   "ComSd".Data.PlcOutputNormal."Q0.0" := "O_14VK1+SGV";
   "ComSd".Data.PlcOutputNormal."Q0.1" := "O_14VK2+SGV";
   "ComSd".Data.PlcOutputNormal."Q0.2" := "O_0VK1+SGV";
   "ComSd".Data.PlcOutputNormal."Q0.3" := "O_0VK2+SGV";
   "ComSd".Data.PlcOutputNormal."Q0.4" := "O_0VK3+SGV";
   "ComSd".Data.PlcOutputNormal."Q0.5" := "O_0VK4+SGV";
   "ComSd".Data.PlcOutputNormal."Q0.6" := "O_0F1.1+SGV";
   "ComSd".Data.PlcOutputNormal."Q0.7" := "O_0KA0.1+SGV";
   "ComSd".Data.PlcOutputNormal."Q1.0" := "O_0KA0.2+SGV";
   "ComSd".Data.PlcOutputNormal."Q1.1" := "O_0KA1+SGV";
   "ComSd".Data.PlcOutputNormal."Q1.2" := "O_8M1.T_c";
   "ComSd".Data.PlcOutputNormal."Q1.3" := "O_8M1.T_o";
   "ComSd".Data.PlcOutputNormal."Q1.4" := "O_8M1.L_c";
   "ComSd".Data.PlcOutputNormal."Q1.5" := "O_8M1.L_o";
   "ComSd".Data.PlcOutputNormal."Q1.6" := "O_8M1.R_c";
   "ComSd".Data.PlcOutputNormal."Q1.7" := "O_8M1.R_o";
   "ComSd".Data.PlcOutputNormal."Q2.0" := "O_8KA1+SGV";
   "ComSd".Data.PlcOutputNormal."Q2.1" := "O_8M1.B_l";
   "ComSd".Data.PlcOutputNormal."Q2.2" := "O_8M1.B_r";
   "ComSd".Data.PlcOutputNormal."Q2.3" := "O_2YV1/2.B+SGV";
   "ComSd".Data.PlcOutputNormal."Q2.4" := "O_2YV1.L+SGV";
   "ComSd".Data.PlcOutputNormal."Q2.5" := "O_2YV1.R+SGV";
   "ComSd".Data.PlcOutputNormal."Q2.6" := "O_5YV1+SGX";
   "ComSd".Data.PlcOutputNormal."Q2.7" := "O_spare27";
END_REGION

REGION Network 4 (SCL): Data PLC Output Safety

   "ComSd".Data.PlcOutputSafety."Q900.0" := "SO_safetynew";
   "ComSd".Data.PlcOutputSafety."Q900.1" := "SO_14HV1+SSTL/R";
   "ComSd".Data.PlcOutputSafety."Q900.2" := "SO_14KA1+SGV";
   "ComSd".Data.PlcOutputSafety."Q900.3" := "SO_14KA2+SGV";
   "ComSd".Data.PlcOutputSafety."Q908.0" := "SO_ST.3HF+SGV";
   "ComSd".Data.PlcOutputSafety."Q908.1" := "SO_ST.5HF+SGV";
   "ComSd".Data.PlcOutputSafety."Q908.2" := "SO_5AX1+SGX";
   "ComSd".Data.PlcOutputSafety."Q908.3" := "SO_spare9083";
END_REGION
END_FUNCTION_BLOCK

FUNCTION_BLOCK "ErrCom"   // FB303, FBD
{ S7_Optimized_Access := 'FALSE' }
// stored: AutoNumber false, SetENOAutomatically false
   VAR
      Var { S7_SetPoint := 'True'} : "TypeVar";
      T : Array[1..1] of IEC_TIMER;
   END_VAR
   VAR_TEMP
      ComOk : Bool;
      PwrOk : Bool;
      SiOk : Bool;
      EsOk : Bool;
      DoorOk : Bool;
   END_VAR
BEGIN

NETWORK
TITLE = general ok
// communication ok
      AN    "G".errComPc;
      =     #ComOk;

// power supply ok
      AN    "G"."errPs-0F1.1+SGV";
      =     #PwrOk;

// safety ok
      AN    "G".errSafetyModules;
      AN    "Si".aLaserErrFdb;
      AN    "Si".aAdjustmentErrFdb1;
      AN    "Si".aAdjustmentErrFdb2;
      =     #SiOk;

// doors ok
      A     #PwrOk;
      A     #SiOk;
      A     "Si".esInternal;
      =     #DoorOk;

// emergency ok
      A     #PwrOk;
      A     #SiOk;
      =     #EsOk;

REGION Network 2 (SCL): emergency stop

   // emergency stop internal (HMI)
   "ComErr".Err[2000] := #EsOk AND NOT "SI_14SB0/1+HMI" AND NOT "I_14SB0+HMI";
   "ComErr".Err[2001] := #EsOk AND NOT "SI_14SB0/1+HMI" AND NOT "I_14SB1+HMI";
   "ComErr".Err[2002] := #EsOk AND "Si".esInternalAckReq;

   // emergency stop external
   "ComErr".Err[2004] := #EsOk AND NOT "SI_NA_EXT+SGV";
   "ComErr".Err[2005] := #EsOk AND "Si".esExternalAckReq;
END_REGION

REGION Network 3 (SCL): safety doors

   // visual measurement - SGV
   "ComErr".Err[2010] := #DoorOk AND NOT "Si"."SGV-14SS1.TL".sig;
   "ComErr".Err[2011] := #DoorOk AND "Si"."SGV-14SS1.TL".sig AND NOT "Si"."SGV-14SS1.TL".ok;

   "ComErr".Err[2013] := #DoorOk AND NOT "Si"."SGV-14SS1.BL".sig;
   "ComErr".Err[2014] := #DoorOk AND "Si"."SGV-14SS1.BL".sig AND NOT "Si"."SGV-14SS1.BL".ok;

   "ComErr".Err[2016] := #DoorOk AND NOT "Si"."SGV-14SS1.TR".sig;
   "ComErr".Err[2017] := #DoorOk AND "Si"."SGV-14SS1.TR".sig AND NOT "Si"."SGV-14SS1.TR".ok;

   "ComErr".Err[2019] := #DoorOk AND NOT "Si"."SGV-14SS1.BR".sig;
   "ComErr".Err[2020] := #DoorOk AND "Si"."SGV-14SS1.BR".sig AND NOT "Si"."SGV-14SS1.BR".ok;

   // visual measurement - SGX
   "ComErr".Err[2030] := #DoorOk AND NOT "Si"."SGX-14SS1.TL".sig;
   "ComErr".Err[2031] := #DoorOk AND "Si"."SGX-14SS1.TL".sig AND NOT "Si"."SGX-14SS1.TL".ok;

   "ComErr".Err[2033] := #DoorOk AND NOT "Si"."SGX-14SS1.BL".sig;
   "ComErr".Err[2034] := #DoorOk AND "Si"."SGX-14SS1.BL".sig AND NOT "Si"."SGX-14SS1.BL".ok;

   "ComErr".Err[2036] := #DoorOk AND NOT "Si"."SGX-14SS1.TR".sig;
   "ComErr".Err[2037] := #DoorOk AND "Si"."SGX-14SS1.TR".sig AND NOT "Si"."SGX-14SS1.TR".ok;

   "ComErr".Err[2039] := #DoorOk AND NOT "Si"."SGX-14SS1.BR".sig;
   "ComErr".Err[2040] := #DoorOk AND "Si"."SGX-14SS1.BR".sig AND NOT "Si"."SGX-14SS1.BR".ok;
END_REGION

REGION Network 4 (SCL): manual

   // setting mode - SSTL
   "ComErr".Err[2050] := #ComOk AND #PwrOk AND #SiOk AND "Si".esInternal AND "Si".settingModeActive;

   // jog mode - SSTL
   "ComErr".Err[2052] := #ComOk AND #PwrOk AND #SiOk AND "Si".esInternal AND "Si".jogModeActive;

   // air-conditioning off - SSTR
   "ComErr".Err[2054] := #ComOk AND #PwrOk AND "I_0SH1+SSTR";
END_REGION

REGION Network 5 (SCL): safety

   // fault safety modules plc
   "ComErr".Err[2060] := #ComOk AND #PwrOk AND "G".errSafetyModules;

   // areas
   "ComErr".Err[2075] := #ComOk AND #PwrOk AND "SI_NA_EXT+SGV" AND  "SI_14SB0/1+HMI" AND (NOT "Si".esInternal OR NOT "Si".esExternal);

   // monitoring feedback
   "ComErr".Err[2080] := #ComOk AND #PwrOk AND "Si".aLaserErrFdb;
   "ComErr".Err[2081] := #ComOk AND #PwrOk AND "Si".aAdjustmentErrFdb1;
   "ComErr".Err[2082] := #ComOk AND #PwrOk AND "Si".aAdjustmentErrFdb2;
   "ComErr".Err[2083] := #ComOk AND #PwrOk AND  "G".Cfg.xrayActive AND "Si".aXrayErrFdb;
END_REGION

REGION Network 6 (SCL): fault sensor
   "ComErr".Err[2090] := "Sen"."1BTR2+SGV".err;
   "ComErr".Err[2091] := "Sen"."1BTR2+SGX".err;
END_REGION

REGION Network 7 (SCL): fault encoder
   "ComErr".Err[2100] := "Enc"."1BCI1".err;
   "ComErr".Err[2101] := "Enc"."1BCM1".err;
   "ComErr".Err[2102] := "Enc"."1BCO1".err;
END_REGION

REGION Network 8 (SCL): communication
   // fault watchdog
   "ComErr".Err[2110] := "G".errComPc;

   // release infeed
   "ComErr".Err[2111] := "G".errNoReleaseInf;
END_REGION

REGION Network 9 (SCL): fault general

   // power supply
   "ComErr".Err[2120] := "G"."errPs-0F1.1+SGV";

   // air conditioner
   "ComErr".Err[2121] := "G"."errAc-0E1+SGV";
   "ComErr".Err[2122] := "G"."errAc-0E2+SGX";
   "ComErr".Err[2123] := "G"."errAc-0E1.1+SGV";

   // err version
   "ComErr".Err[2125] := "G".errVersion;
END_REGION

REGION Network 10 (SCL): off information
   "ComErr".Err[2140] := "G".adjScannerOff;
   "ComErr".Err[2141] := "G".adjTopOff;
   "ComErr".Err[2142] := "G".adjLeftOff;
   "ComErr".Err[2143] := "G".adjRightOff;
   "ComErr".Err[2144] := "G".air1Off;
   "ComErr".Err[2145] := "G".air2Off;
   "ComErr".Err[2146] := "G".airXrayOff;
   "ComErr".Err[2147] := "G".airDehOff;
END_REGION

REGION Network 11 (SCL): fault adjustment

   // adjustment scannerhousing (-8M1.B+SGV)
   "ComErr".Err[2150] := "ComSd".Data.Scanner.Err;
   "ComErr".Err[2151] := "Enc"."8B1.B".err;
   "ComErr".Err[2152] := "Sen"."8S1.B".err;
   "ComErr".Err[2153] := "Sen"."8S2.B".err;
   "ComErr".Err[2154] := "Si".aAdjustment AND NOT "ComSd".Data.Scanner.refRun AND NOT "ComSd".Data.Scanner.refOk;
   "ComErr".Err[2155] := "Si".aAdjustment AND "ComSd".Data.Scanner.refRun;
   "ComErr".Err[2156] := "Si".aAdjustment AND "AdjScanner_DB".Cmd.auto AND NOT"ComSd".Data.Scanner.PosOk;
   "ComErr".Err[2157] := "Si".aAdjustment AND "ComRd".Data.Scanner.ManModeActive;

   // adjustment metering bar top (-8M1.T+SGV)
   "ComErr".Err[2160] := "ComSd".Data.Top.Err;
   "ComErr".Err[2161] := "ComSd".Data.Top.ErrEnc;
   "ComErr".Err[2162] := "Sen"."8S1.T".err;
   "ComErr".Err[2163] := "Sen"."8S2.T".err;
   "ComErr".Err[2164] := "Si".aAdjustment AND NOT "ComSd".Data.Top.refRun AND NOT "ComSd".Data.Top.refOk;
   "ComErr".Err[2165] := "Si".aAdjustment AND "ComSd".Data.Top.refRun;
   "ComErr".Err[2166] := "Si".aAdjustment AND "AdjTop_DB".Cmd.auto AND ((NOT "G".Cfg.adjTopActiveLinMot AND "Enc"."8BC1.T".notInPos) OR ("G".Cfg.adjTopActiveLinMot AND "Enc"."8U1.T".notInPos));
   "ComErr".Err[2167] := "Si".aAdjustment AND "ComRd".Data.Top.ManModeActive;

   // adjustment metering bar left (-8M1.L+SGV)
   "ComErr".Err[2170] := "ComSd".Data.Left.Err;
   "ComErr".Err[2171] := "ComSd".Data.Left.ErrEnc;
   "ComErr".Err[2172] := "Sen"."8S1.L".err;
   "ComErr".Err[2173] := "Sen"."8S2.L".err;
   "ComErr".Err[2174] := "Si".aAdjustment AND NOT "ComSd".Data.Left.refRun AND NOT "ComSd".Data.Left.refOk;
   "ComErr".Err[2175] := "Si".aAdjustment AND "ComSd".Data.Left.refRun;
   "ComErr".Err[2176] := "Si".aAdjustment AND "AdjLeft_DB".Cmd.auto AND ((NOT "G".Cfg.adjLeftActiveLinMot AND "Enc"."8BC1.L".notInPos) OR ("G".Cfg.adjLeftActiveLinMot AND "Enc"."8U1.L".notInPos));
   "ComErr".Err[2177] := "Si".aAdjustment AND "ComRd".Data.Left.ManModeActive;

   // adjustment metering bar right (-8M1.R+SGV)
   "ComErr".Err[2180] := "ComSd".Data.Right.Err;
   "ComErr".Err[2181] := "ComSd".Data.Right.ErrEnc;
   "ComErr".Err[2182] := "Sen"."8S1.R".err;
   "ComErr".Err[2183] := "Sen"."8S2.R".err;
   "ComErr".Err[2184] := "Si".aAdjustment AND NOT "ComSd".Data.Right.refRun AND NOT "ComSd".Data.Right.refOk;
   "ComErr".Err[2185] := "Si".aAdjustment AND "ComSd".Data.Right.refRun;
   "ComErr".Err[2186] := "Si".aAdjustment AND "AdjRight_DB".Cmd.auto AND ((NOT "G".Cfg.adjRightActiveLinMot AND "Enc"."8BC1.R".notInPos) OR ("G".Cfg.adjRightActiveLinMot AND "Enc"."8U1.R".notInPos));
   "ComErr".Err[2187] := "Si".aAdjustment AND "ComRd".Data.Right.ManModeActive;

   // sensor for random adjustment
   "ComErr".Err[2190] := "Sen"."8B1".err AND "G".Cfg.adjTopActiveLinMot;
   "ComErr".Err[2191] := "Sen"."8B2".err AND "G".Cfg.adjLeftActiveLinMot;
   "ComErr".Err[2192] := "Sen"."8B3".err AND "G".Cfg.adjRightActiveLinMot;
END_REGION

REGION Network 12 (SCL): fault profinet

   // fault profinet
   "ComErr".Err[2200] := "Diag_DB".IoDataSys1.devices[1].error AND "G".Cfg.adjTopActiveLinMot;
   "ComErr".Err[2201] := "Diag_DB".IoDataSys1.devices[2].error AND "G".Cfg.adjLeftActiveLinMot;
   "ComErr".Err[2202] := "Diag_DB".IoDataSys1.devices[3].error AND "G".Cfg.adjRightActiveLinMot;
END_REGION
END_FUNCTION_BLOCK

FUNCTION_BLOCK "DataTakeOver"   // FB302, FBD
{ S7_Optimized_Access := 'TRUE' }
// stored: AutoNumber false, MemoryReserve 100, SetENOAutomatically false
   VAR
      Var { ExternalAccessible := 'False'; ExternalVisible := 'False'; ExternalWritable := 'False'} : "TypeVar";
   END_VAR
BEGIN

REGION Network 1 (SCL): config data from pc
   IF "ComRd".Data.Config.active AND "G".comOk THEN

       // config for mode
       "G".Cfg.adjScannerActive := "ComRd".Data.Config.adjScannerActive;
       "G".Cfg.adjTopActive := "ComRd".Data.Config.adjTopActive;
       "G".Cfg.adjLeftActive := "ComRd".Data.Config.adjLeftActive;
       "G".Cfg.adjRightActive := "ComRd".Data.Config.adjRightActive;

       "G".Cfg.adjTopActiveLinMot := "ComRd".Data.Config.adjTopLinMotActive;
       "G".Cfg.adjLeftActiveLinMot := "ComRd".Data.Config.adjLeftLinMotActive;
       "G".Cfg.adjRightActiveLinMot := "ComRd".Data.Config.adjRightLinMotActive;

       "G".Cfg.xrayActive := "ComRd".Data.Config.xrayActive ;

       // config for mode
       "G".Cfg.modeBoardPassing:= "ComRd".Data.Config.modeBoardPassing;
       "G".Cfg.modeDimension := "ComRd".Data.Config.modeDimension;
       "G".Cfg.modeRandomAdj := "ComRd".Data.Config.modeRandomAdj;

       // config for sensor for random adjustment
       IF "ComRd".Data.Config.modeDimension = 3 OR "ComRd".Data.Config.modeDimension = 4 THEN
           "G".Cfg.senTopActive := TRUE;
       ELSE
           "G".Cfg.senTopActive := FALSE;
       END_IF;
       IF "ComRd".Data.Config.modeDimension = 2 OR "ComRd".Data.Config.modeDimension = 4 THEN
           IF "ComRd".Data.Config.modeBoardPassing = 3 THEN
               "G".Cfg.senLeftActive := TRUE;
               "G".Cfg.senRightActive := TRUE;
           ELSIF "ComRd".Data.Config.modeBoardPassing = 2 THEN
               "G".Cfg.senLeftActive := TRUE;
               "G".Cfg.senRightActive := FALSE;
           ELSIF "ComRd".Data.Config.modeBoardPassing = 1 THEN
               "G".Cfg.senLeftActive := FALSE;
               "G".Cfg.senRightActive := TRUE;
           END_IF;
       ELSE
           "G".Cfg.senLeftActive := FALSE;
           "G".Cfg.senRightActive := FALSE;
       END_IF;

       // config for encoder 1
       IF "ComRd".Data.Config.enc1QuadEvalActive THEN
           "G".Cfg.enc1Gain := (1.0 / INT_TO_REAL("ComRd".Data.Config.enc1Factor)) * 1.0;
       ELSE
           "G".Cfg.enc1Gain := (1.0 / INT_TO_REAL("ComRd".Data.Config.enc1Factor)) * 1.0;
       END_IF;
       IF "ComRd".Data.Config.enc1Factor = -1 THEN
           "G".Cfg.enc1Active := FALSE;
       ELSE
           "G".Cfg.enc1Active := TRUE;
       END_IF;

   END_IF;
END_REGION

REGION Network 2 (SCL): batch from pc
   IF "G".comOk THEN
       // Width
       IF "ComRd".Data.batch.MinWidth = "ComRd".Data.batch.MaxWidth THEN
           "G".Batch.widthMin := DINT_TO_REAL("ComRd".Data.batch.MinWidth) / 10.0;
           "G".Batch.widthMax := DINT_TO_REAL("ComRd".Data.batch.MaxWidth) / 10.0;
           "G".Batch.width := DINT_TO_REAL("ComRd".Data.batch.MinWidth) / 10.0;
       ELSIF "ComRd".Data.batch.MinWidth <> "ComRd".Data.batch.MaxWidth THEN
           "G".Batch.widthMin := DINT_TO_REAL("ComRd".Data.batch.MinWidth) / 10.0;
           "G".Batch.widthMax := DINT_TO_REAL("ComRd".Data.batch.MaxWidth) / 10.0;
           "G".Batch.width := DINT_TO_REAL(("ComRd".Data.batch.MinWidth + "ComRd".Data.batch.MaxWidth) / 2) / 10.0;
       END_IF;

       // Thickness
       IF "ComRd".Data.batch.MinThickness = "ComRd".Data.batch.MaxThickness THEN
           "G".Batch.thicknessMin := DINT_TO_REAL("ComRd".Data.batch.MinThickness) / 10.0;
           "G".Batch.thicknessMax := DINT_TO_REAL("ComRd".Data.batch.MaxThickness) / 10.0;
           "G".Batch.thickness := DINT_TO_REAL("ComRd".Data.batch.MinThickness) / 10.0;
       ELSIF "ComRd".Data.batch.MinThickness <> "ComRd".Data.batch.MaxThickness THEN
           "G".Batch.thicknessMin := DINT_TO_REAL("ComRd".Data.batch.MinThickness) / 10.0;
           "G".Batch.thicknessMax := DINT_TO_REAL("ComRd".Data.batch.MaxThickness) / 10.0;
           "G".Batch.thickness := DINT_TO_REAL(("ComRd".Data.batch.MinThickness + "ComRd".Data.batch.MaxThickness) / 2) / 10.0;
       END_IF;
   END_IF;
END_REGION
END_FUNCTION_BLOCK

FUNCTION_BLOCK "Sensors"   // FB505, FBD
{ S7_Optimized_Access := 'TRUE' }
// stored: AutoNumber false, MemoryReserve 100, SetENOAutomatically false
   VAR
      Var { ExternalAccessible := 'False'; ExternalVisible := 'False'; ExternalWritable := 'False'} : "TypeVar";
      Enc { ExternalAccessible := 'False'; ExternalVisible := 'False'; ExternalWritable := 'False'} : Array[1..3] of "SysCounterFast";
      S { ExternalAccessible := 'False'; ExternalVisible := 'False'; ExternalWritable := 'False'} : Array[1..5] of "SysSensor";
      SIO { ExternalAccessible := 'False'; ExternalVisible := 'False'; ExternalWritable := 'False'} : Array[1..3] of "SysWenglorP3PC301";
      senRightEncAct { ExternalAccessible := 'False'; ExternalVisible := 'False'; ExternalWritable := 'False'} : Real;
      senRightValSmoth { ExternalAccessible := 'False'; ExternalVisible := 'False'; ExternalWritable := 'False'} : Real;
      senRightCntr { ExternalAccessible := 'False'; ExternalVisible := 'False'; ExternalWritable := 'False'} : DInt;
      senRightSum { ExternalAccessible := 'False'; ExternalVisible := 'False'; ExternalWritable := 'False'} : Real;
      senLeftEncAct { ExternalAccessible := 'False'; ExternalVisible := 'False'; ExternalWritable := 'False'} : Real;
      senLeftValSmoth { ExternalAccessible := 'False'; ExternalVisible := 'False'; ExternalWritable := 'False'} : Real;
      senLeftCntr { ExternalAccessible := 'False'; ExternalVisible := 'False'; ExternalWritable := 'False'} : DInt;
      senLeftSum { ExternalAccessible := 'False'; ExternalVisible := 'False'; ExternalWritable := 'False'} : Real;
      senTopEncAct { ExternalAccessible := 'False'; ExternalVisible := 'False'; ExternalWritable := 'False'} : Real;
      senTopValSmoth { ExternalAccessible := 'False'; ExternalVisible := 'False'; ExternalWritable := 'False'} : Real;
      senTopCntr { ExternalAccessible := 'False'; ExternalVisible := 'False'; ExternalWritable := 'False'} : DInt;
      senTopSum { ExternalAccessible := 'False'; ExternalVisible := 'False'; ExternalWritable := 'False'} : Real;
      deltaSaved { ExternalAccessible := 'False'; ExternalVisible := 'False'; ExternalWritable := 'False'} : Real;
      senLeftValValid { ExternalAccessible := 'False'; ExternalVisible := 'False'; ExternalWritable := 'False'} : Bool;
      senRightValValid { ExternalAccessible := 'False'; ExternalVisible := 'False'; ExternalWritable := 'False'} : Bool;
      senTopValValid { ExternalAccessible := 'False'; ExternalVisible := 'False'; ExternalWritable := 'False'} : Bool;
      widthMeasureOk { ExternalAccessible := 'False'; ExternalVisible := 'False'; ExternalWritable := 'False'} : Bool;
   END_VAR
   VAR_TEMP
      tempMin : Real;
      tempMax : Real;
      tempWidth : Real;
   END_VAR
   VAR_TEMP   // added for the SCL form of the ladder/FBD networks
      _w1 : Bool;
   END_VAR
BEGIN

REGION Network 1: encoder infeed scanner
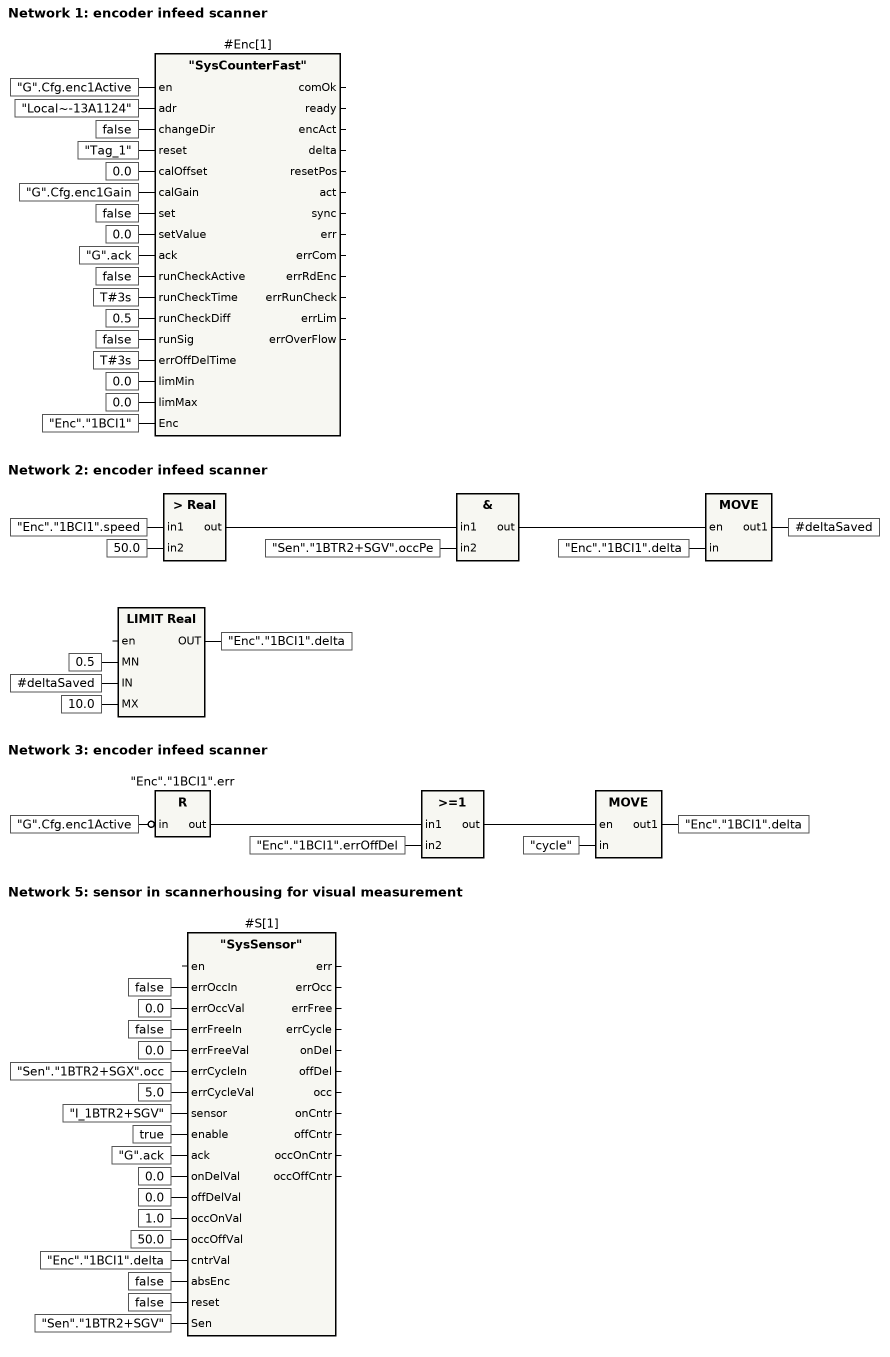
   IF "G".Cfg.enc1Active THEN
       #Enc[1](adr := "Local~-13A1124",   // "SysCounterFast"
               changeDir := false,
               reset := "Tag_1",
               calOffset := 0.0,
               calGain := "G".Cfg.enc1Gain,
               set := false,
               setValue := 0.0,
               ack := "G".ack,
               runCheckActive := false,
               runCheckTime := T#3s,
               runCheckDiff := 0.5,
               runSig := false,
               errOffDelTime := T#3s,
               limMin := 0.0,
               limMax := 0.0,
               Enc := "Enc"."1BCI1");
   END_IF;
END_REGION

REGION Network 2: encoder infeed scanner
   IF ("Enc"."1BCI1".speed > 50.0) AND "Sen"."1BTR2+SGV".occPe THEN
       #deltaSaved := "Enc"."1BCI1".delta;
   END_IF;
   "Enc"."1BCI1".delta := LIMIT(MN := 0.5, IN := #deltaSaved, MX := 10.0);
END_REGION

REGION Network 3: encoder infeed scanner
   IF NOT "G".Cfg.enc1Active THEN "Enc"."1BCI1".err := FALSE; END_IF;
   IF NOT "G".Cfg.enc1Active OR "Enc"."1BCI1".errOffDel THEN "Enc"."1BCI1".delta := "cycle"; END_IF;
END_REGION

REGION Network 4: - sensor monitoring -
END_REGION

REGION Network 5: sensor in scannerhousing for visual measurement
   #S[1](errOccIn := false,   // "SysSensor"
         errOccVal := 0.0,
         errFreeIn := false,
         errFreeVal := 0.0,
         errCycleIn := "Sen"."1BTR2+SGX".occ,
         errCycleVal := 5.0,
         sensor := "I_1BTR2+SGV",
         enable := true,
         ack := "G".ack,
         onDelVal := 0.0,
         offDelVal := 0.0,
         occOnVal := 1.0,
         occOffVal := 50.0,
         cntrVal := "Enc"."1BCI1".delta,
         absEnc := false,
         reset := false,
         Sen := "Sen"."1BTR2+SGV");
END_REGION

REGION Network 6: sensor in scannerhousing for xray measurement
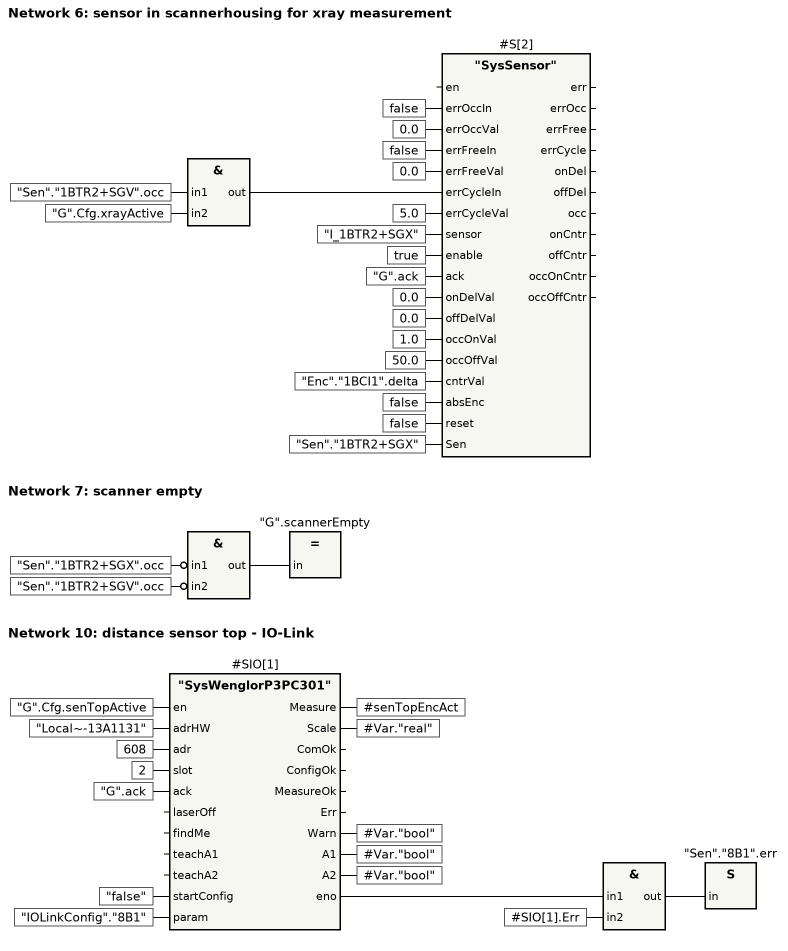
   #S[2](errOccIn := false,   // "SysSensor"
         errOccVal := 0.0,
         errFreeIn := false,
         errFreeVal := 0.0,
         errCycleIn := "Sen"."1BTR2+SGV".occ AND "G".Cfg.xrayActive,
         errCycleVal := 5.0,
         sensor := "I_1BTR2+SGX",
         enable := true,
         ack := "G".ack,
         onDelVal := 0.0,
         offDelVal := 0.0,
         occOnVal := 1.0,
         occOffVal := 50.0,
         cntrVal := "Enc"."1BCI1".delta,
         absEnc := false,
         reset := false,
         Sen := "Sen"."1BTR2+SGX");
END_REGION

REGION Network 7: scanner empty
   "G".scannerEmpty := NOT "Sen"."1BTR2+SGX".occ AND NOT "Sen"."1BTR2+SGV".occ;
END_REGION

REGION Network 8: distance sensor top
END_REGION

REGION Network 9 (SCL): distance sensor top - calibration value from pc
   "ComSd".Data.Measure.SetCalibratePosTopOk := FALSE;

   IF "ComRd".Data.Measure.SetCalibratePosTop THEN

       "Ref".senTopCalOffset := #senTopEncAct + "G".Batch.thickness;
       "ComSd".Data.Measure.SetCalibratePosTopOk := TRUE;
   END_IF;
END_REGION

REGION Network 10: distance sensor top - IO-Link
   #SIO[1](EN := "G".Cfg.senTopActive,   // "SysWenglorP3PC301"
           adrHW := "Local~-13A1131",
           adr := 608,
           slot := 2,
           ack := "G".ack,
           startConfig := "false",
           param := "IOLinkConfig"."8B1",
           Measure => #senTopEncAct,
           Scale => #Var."real",
           Warn => #Var."bool",
           A1 => #Var."bool",
           A2 => #Var."bool",
           ENO => #_w1);
   IF #_w1 AND #SIO[1].Err THEN "Sen"."8B1".err := TRUE; END_IF;
END_REGION

REGION Network 11 (SCL): distance sensor top - values
   IF "G".Cfg.senTopActive THEN
       IF #SIO[1].MeasureOk THEN
           "Sen"."8B1".val := "Ref".senTopCalOffset - #senTopEncAct;
       ELSE
           "Sen"."8B1".val := -50.0;
       END_IF;
       "ComSd".Data.Measure.ActValueTop := REAL_TO_DINT(#senTopEncAct * 10.0);

       IF "G".Cfg.modeBoardPassing = 3 THEN
           #tempMin := "G".Batch.widthMin / 4.0;
           #tempMax := "G".Batch.widthMax + 50.0;
       ELSE
           #tempMin := "G".Batch.widthMin / 2.0;
           #tempMax := "G".Batch.widthMax + 50.0;
       END_IF;
   ELSE
       #senTopEncAct :=  "Sen"."8B1".val := 0.0;
       "ComSd".Data.Measure.ActValueTop := 0;
   END_IF;
END_REGION

REGION Network 12: distance sensor top - occupied
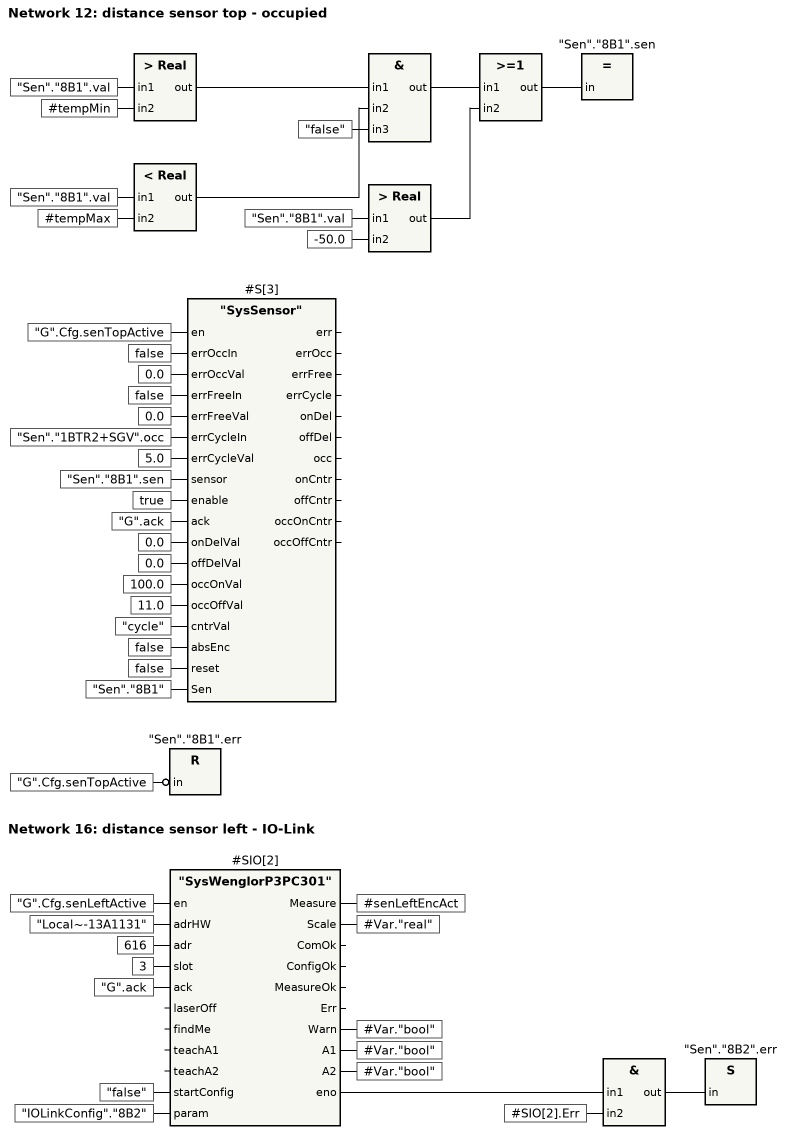
   "Sen"."8B1".sen := (("Sen"."8B1".val > #tempMin) AND ("Sen"."8B1".val < #tempMax) AND "false") OR ("Sen"."8B1".val > (-50.0));
   IF "G".Cfg.senTopActive THEN
       #S[3](errOccIn := false,   // "SysSensor"
             errOccVal := 0.0,
             errFreeIn := false,
             errFreeVal := 0.0,
             errCycleIn := "Sen"."1BTR2+SGV".occ,
             errCycleVal := 5.0,
             sensor := "Sen"."8B1".sen,
             enable := true,
             ack := "G".ack,
             onDelVal := 0.0,
             offDelVal := 0.0,
             occOnVal := 100.0,
             occOffVal := 11.0,
             cntrVal := "cycle",
             absEnc := false,
             reset := false,
             Sen := "Sen"."8B1");
   END_IF;
   IF NOT "G".Cfg.senTopActive THEN "Sen"."8B1".err := FALSE; END_IF;
END_REGION

REGION Network 13 (SCL): distance sensor top - smoothed value
   IF "Sen"."8B1".occPe THEN
       #senTopCntr := 10;
       #senTopSum := 0.0;
       #senTopValValid := false;
   ELSIF NOT "Sen"."8B1".occ OR #senTopCntr > 10 THEN
       #senTopCntr := 0;
   END_IF;

   IF "Sen"."8B1".occNe THEN
       #senTopValValid := false;
   END_IF;

   IF #senTopCntr > 0 AND "Sen"."8B1".sen THEN
       #senTopSum += "Sen"."8B1".val;
       #senTopCntr -= 1;
       IF #senTopCntr = 0 THEN
           #senTopValSmoth := #senTopSum / 10.0;
           #senTopValValid := true;
       END_IF;
   END_IF;

   IF "ComRd".Data.status.Auto AND  "G".Cfg.senTopActive THEN
       "Sen"."8B1".val := #senTopValSmoth;
   END_IF;
END_REGION

REGION Network 14: distance sensor left
END_REGION

REGION Network 15 (SCL): distance sensor left - calibration value from pc
   "ComSd".Data.Measure.SetCalibratePosLeftOk := FALSE;

   IF "ComRd".Data.Measure.SetCalibratePosLeft THEN

       #tempWidth := "G".Batch.width;
       IF "G".Cfg.modeBoardPassing = 3 THEN
           #tempWidth := "G".Batch.width / 2.0;
       END_IF;
       "Ref".senLeftCalOffset := #senLeftEncAct + #tempWidth;

       "ComSd".Data.Measure.SetCalibratePosLeftOk := TRUE;
   END_IF;
END_REGION

REGION Network 16: distance sensor left - IO-Link
   #SIO[2](EN := "G".Cfg.senLeftActive,   // "SysWenglorP3PC301"
           adrHW := "Local~-13A1131",
           adr := 616,
           slot := 3,
           ack := "G".ack,
           startConfig := "false",
           param := "IOLinkConfig"."8B2",
           Measure => #senLeftEncAct,
           Scale => #Var."real",
           Warn => #Var."bool",
           A1 => #Var."bool",
           A2 => #Var."bool",
           ENO => #_w1);
   IF #_w1 AND #SIO[2].Err THEN "Sen"."8B2".err := TRUE; END_IF;
END_REGION

REGION Network 17 (SCL): distance sensor left - values
   IF "G".Cfg.senLeftActive THEN

       IF #SIO[2].MeasureOk THEN
           "Sen"."8B2".val := "Ref".senLeftCalOffset - #senLeftEncAct;
       ELSE
           "Sen"."8B2".val := -50.0;
       END_IF;
       "ComSd".Data.Measure.ActValueLeft := REAL_TO_DINT("Sen"."8B2".val * 10.0);

       IF "G".Cfg.modeBoardPassing = 3 THEN
           #tempMin := "G".Batch.widthMin / 4.0;
           #tempMax := "G".Batch.widthMax + 50.0;
       ELSE
           #tempMin := "G".Batch.widthMin / 2.0;
           #tempMax := "G".Batch.widthMax + 50.0;
       END_IF;
   ELSE
       #senLeftEncAct :=  "Sen"."8B2".val := 0.0;
       "ComSd".Data.Measure.ActValueLeft := 0;
   END_IF;
END_REGION

REGION Network 18: distance sensor left - occupied
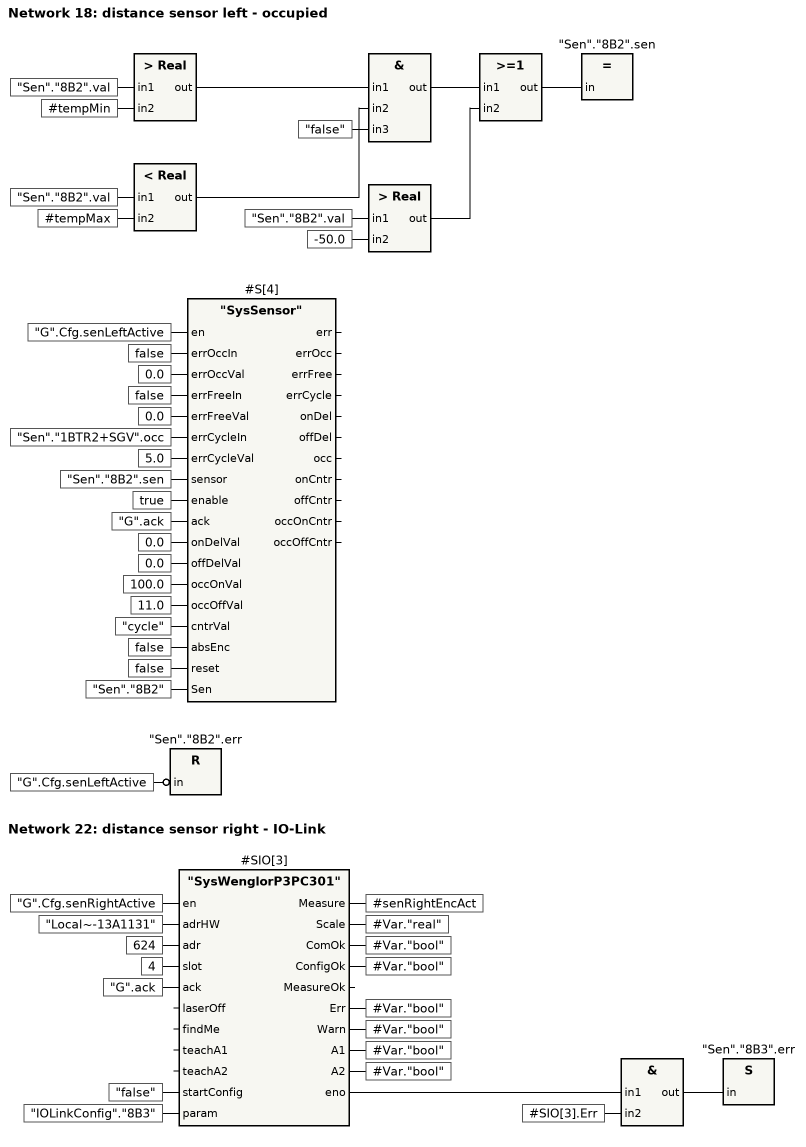
   "Sen"."8B2".sen := (("Sen"."8B2".val > #tempMin) AND ("Sen"."8B2".val < #tempMax) AND "false") OR ("Sen"."8B2".val > (-50.0));
   IF "G".Cfg.senLeftActive THEN
       #S[4](errOccIn := false,   // "SysSensor"
             errOccVal := 0.0,
             errFreeIn := false,
             errFreeVal := 0.0,
             errCycleIn := "Sen"."1BTR2+SGV".occ,
             errCycleVal := 5.0,
             sensor := "Sen"."8B2".sen,
             enable := true,
             ack := "G".ack,
             onDelVal := 0.0,
             offDelVal := 0.0,
             occOnVal := 100.0,
             occOffVal := 11.0,
             cntrVal := "cycle",
             absEnc := false,
             reset := false,
             Sen := "Sen"."8B2");
   END_IF;
   IF NOT "G".Cfg.senLeftActive THEN "Sen"."8B2".err := FALSE; END_IF;
END_REGION

REGION Network 19 (SCL): distance sensor left - smoothed value
   IF "Sen"."8B2".occPe THEN
       #senLeftCntr := 10;
       #senLeftSum := 0.0;
       #senLeftValValid := false;
   ELSIF NOT "Sen"."8B2".occ OR #senLeftCntr > 10 THEN
       #senLeftCntr := 0;
   END_IF;

   IF "Sen"."8B2".occNe THEN
       #senLeftValValid := false;
   END_IF;

   IF #senLeftCntr > 0 AND "Sen"."8B2".sen THEN
       #senLeftSum += "Sen"."8B2".val;
       #senLeftCntr -= 1;
       IF #senLeftCntr = 0 THEN
           #senLeftValSmoth := #senLeftSum / 10.0;
           #senLeftValValid := true;
       END_IF;
   END_IF;

   IF "ComRd".Data.status.Auto AND  "G".Cfg.senLeftActive THEN
       "Sen"."8B2".val := #senLeftValSmoth;
   END_IF;
END_REGION

REGION Network 20: distance sensor right
END_REGION

REGION Network 21 (SCL): distance sensor right - calibration value from pc
   "ComSd".Data.Measure.SetCalibratePosRightOk := FALSE;

   IF "ComRd".Data.Measure.SetCalibratePosRight THEN

       #tempWidth := "G".Batch.width;
       IF "G".Cfg.modeBoardPassing = 3 THEN
           #tempWidth := "G".Batch.width / 2.0;
       END_IF;
       "Ref".senRightCalOffset := #senRightEncAct + #tempWidth;

       "ComSd".Data.Measure.SetCalibratePosRightOk := TRUE;
   END_IF;
END_REGION

REGION Network 22: distance sensor right - IO-Link
   #SIO[3](EN := "G".Cfg.senRightActive,   // "SysWenglorP3PC301"
           adrHW := "Local~-13A1131",
           adr := 624,
           slot := 4,
           ack := "G".ack,
           startConfig := "false",
           param := "IOLinkConfig"."8B3",
           Measure => #senRightEncAct,
           Scale => #Var."real",
           ComOk => #Var."bool",
           ConfigOk => #Var."bool",
           Err => #Var."bool",
           Warn => #Var."bool",
           A1 => #Var."bool",
           A2 => #Var."bool",
           ENO => #_w1);
   IF #_w1 AND #SIO[3].Err THEN "Sen"."8B3".err := TRUE; END_IF;
END_REGION

REGION Network 23 (SCL): distance sensor right - values
   IF "G".Cfg.senRightActive THEN
       IF #SIO[3].MeasureOk THEN
           "Sen"."8B3".val := "Ref".senRightCalOffset - #senRightEncAct;
       ELSE
           "Sen"."8B3".val := -50.0;
       END_IF;
       "ComSd".Data.Measure.ActValueRight := REAL_TO_DINT("Sen"."8B3".val * 10.0);

       IF "G".Cfg.modeBoardPassing = 3 THEN
           #tempMin := "G".Batch.widthMin / 4.0;
           #tempMax := "G".Batch.widthMax + 50.0;
       ELSE
           #tempMin := "G".Batch.widthMin / 2.0;
           #tempMax := "G".Batch.widthMax + 50.0;
       END_IF;
   ELSE
       #senRightEncAct :=  "Sen"."8B3".val := 0.0;
       "ComSd".Data.Measure.ActValueRight := 0;
   END_IF;
END_REGION

REGION Network 24: distance sensor right - occupied
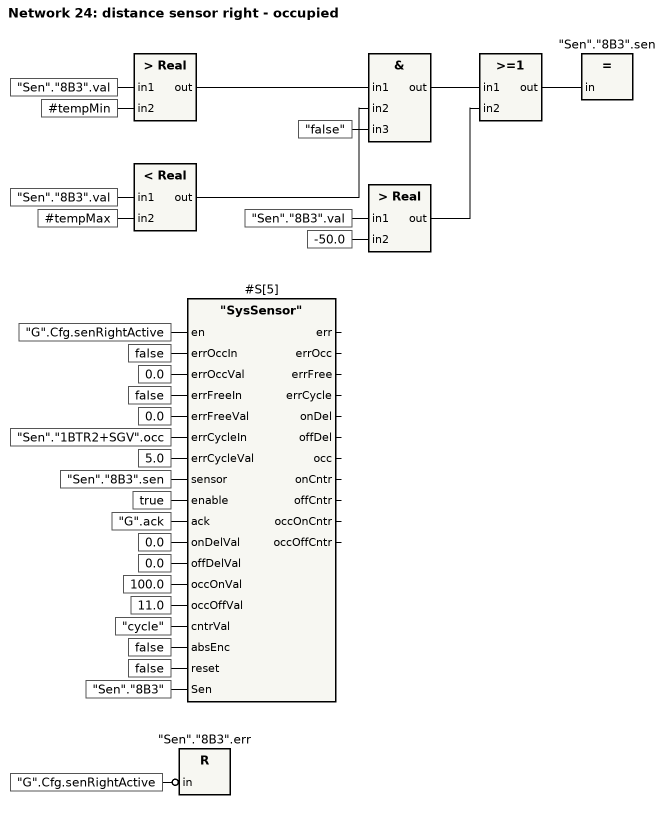
   "Sen"."8B3".sen := (("Sen"."8B3".val > #tempMin) AND ("Sen"."8B3".val < #tempMax) AND "false") OR ("Sen"."8B3".val > (-50.0));
   IF "G".Cfg.senRightActive THEN
       #S[5](errOccIn := false,   // "SysSensor"
             errOccVal := 0.0,
             errFreeIn := false,
             errFreeVal := 0.0,
             errCycleIn := "Sen"."1BTR2+SGV".occ,
             errCycleVal := 5.0,
             sensor := "Sen"."8B3".sen,
             enable := true,
             ack := "G".ack,
             onDelVal := 0.0,
             offDelVal := 0.0,
             occOnVal := 100.0,
             occOffVal := 11.0,
             cntrVal := "cycle",
             absEnc := false,
             reset := false,
             Sen := "Sen"."8B3");
   END_IF;
   IF NOT "G".Cfg.senRightActive THEN "Sen"."8B3".err := FALSE; END_IF;
END_REGION

REGION Network 25 (SCL): distance sensor right - smoothed value
   IF "Sen"."8B3".occPe THEN
       #senRightCntr := 10;
       #senRightSum := 0.0;
       #senRightValValid := false;
   ELSIF NOT "Sen"."8B3".occ OR #senRightCntr > 10 THEN
       #senRightCntr := 0;
   END_IF;

   IF "Sen"."8B3".occNe THEN
       #senRightValValid := false;
   END_IF;

   IF #senRightCntr > 0 AND "Sen"."8B3".sen THEN
       #senRightSum += "Sen"."8B3".val;
       #senRightCntr -= 1;
       IF #senRightCntr = 0 THEN
           #senRightValSmoth := #senRightSum / 10.0;
           #senRightValValid := true;
       END_IF;
   END_IF;

   IF "ComRd".Data.status.Auto AND  "G".Cfg.senRightActive THEN
       "Sen"."8B3".val := #senRightValSmoth;
   END_IF;
END_REGION

REGION Network 26 (SCL): distance sensor - data to pc
   // Thickness
   IF "G".Cfg.modeDimension = 3 OR "G".Cfg.modeDimension = 4 AND  NOT "Sen"."1BTR2+SGV".occ THEN
       "G".Batch.thicknessMeasure := "Sen"."8B1".val;
       // Version 5.13 - Dont look at min or max
       // IF "G".Batch.thicknessMeasure < "G".Batch.thicknessMin OR "G".Batch.thicknessMeasure > "G".Batch.thicknessMax  THEN
       //     "G".Batch.thicknessMeasure := "G".Batch.thickness;
       // END_IF;
       "ComSd".Data.Measure.Thickness := REAL_TO_DINT("G".Batch.thicknessMeasure * 10.0);
   ELSE
       "ComSd".Data.Measure.Thickness := 0;
   END_IF;

   // Width
   IF "G".Cfg.modeDimension = 2 OR "G".Cfg.modeDimension = 4 AND NOT "Sen"."1BTR2+SGV".occ  THEN
       #widthMeasureOk := false;
       IF "G".Cfg.modeBoardPassing = 1 AND  #senRightValValid  THEN
           "G".Batch.widthMeasure := "Sen"."8B3".val;
           #widthMeasureOk := true;
       ELSIF "G".Cfg.modeBoardPassing = 2 AND  #senLeftValValid THEN
           "G".Batch.widthMeasure := "Sen"."8B2".val;
           #widthMeasureOk := true;
       ELSIF "G".Cfg.modeBoardPassing = 3  AND #senLeftValValid  AND #senRightValValid  THEN
           "G".Batch.senLeftVal := "Sen"."8B2".val;
           "G".Batch.senRightVal := "Sen"."8B3".val;
           #widthMeasureOk := true;
           // Version 5.13 - Dont look at min or max
           // IF "G".Batch.senLeftVal < "G".Batch.widthMin / 2.0 - 50.0 OR "G".Batch.senLeftVal > "G".Batch.widthMax / 2.0 + 50.0 OR
           //     "G".Batch.senRightVal < "G".Batch.widthMin / 2.0 - 50.0 OR "G".Batch.senRightVal > "G".Batch.widthMax / 2.0 + 50.0 THEN
           //     "G".Batch.senLeftVal := "G".Batch.senRightVal := "G".Batch.width / 2.0;
           //     #widthMeasureOk := false;
           // END_IF;
           "G".Batch.widthMeasure := "G".Batch.senLeftVal + "G".Batch.senRightVal;
           "G".Batch.offsetBoard := ("G".Batch.senLeftVal - "G".Batch.senRightVal) / 2.0;
       END_IF;
       // Version 5.13 - Dont look at min or max
       // IF "G".Batch.widthMeasure < ("G".Batch.widthMin - 50.0)  OR "G".Batch.widthMeasure > ("G".Batch.widthMax + 50.0) THEN
       //     "G".Batch.widthMeasure := "G".Batch.width;
       //     #widthMeasureOk := false;
       // END_IF;
       "ComSd".Data.Measure.Width := REAL_TO_DINT(("G".Batch.widthMeasure) * 10.0);
   ELSE
       "ComSd".Data.Measure.Width := 0;
   END_IF;
END_REGION
END_FUNCTION_BLOCK

FUNCTION_BLOCK "SysCounterFast"   // FB2035, FBD
TITLE = manage a incremental encoder conected to a counter module
{ S7_Optimized_Access := 'TRUE' }
AUTHOR : MiCROTEC
VERSION : 1.6
// -2018.09 : Martin
// -2019.10 : Martin
// stored: AutoNumber false, MemoryReserve 100, SetENOAutomatically false
   VAR_INPUT
      adr { ExternalAccessible := 'False'; ExternalVisible := 'False'; ExternalWritable := 'False'} : HW_IO;   // I/O adresse
      changeDir { ExternalAccessible := 'False'; ExternalVisible := 'False'; ExternalWritable := 'False'} : Bool;   // change direction
      reset { ExternalAccessible := 'False'; ExternalVisible := 'False'; ExternalWritable := 'False'} : Bool;   // reset counter
      calOffset { ExternalAccessible := 'False'; ExternalVisible := 'False'; ExternalWritable := 'False'} : Real;   // offset [mm], the "Reset" will take effect after the offset value
      calGain { ExternalAccessible := 'False'; ExternalVisible := 'False'; ExternalWritable := 'False'} : Real;   // gain
      set { ExternalAccessible := 'False'; ExternalVisible := 'False'; ExternalWritable := 'False'} : Bool;   // set counter on "set value"
      setValue { ExternalAccessible := 'False'; ExternalVisible := 'False'; ExternalWritable := 'False'} : Real;   // set value [mm]
      ack { ExternalAccessible := 'False'; ExternalVisible := 'False'; ExternalWritable := 'False'} : Bool;   // fault acknowledge
      runCheckActive { ExternalAccessible := 'False'; ExternalVisible := 'False'; ExternalWritable := 'False'} : Bool;   // activate plausibility check of encoder value and run signal
      runCheckTime { ExternalAccessible := 'False'; ExternalVisible := 'False'; ExternalWritable := 'False'} : Time := T#3S;   // run signal check fault time
      runCheckDiff { ExternalAccessible := 'False'; ExternalVisible := 'False'; ExternalWritable := 'False'} : Real := 0.5;   // difference value for run check
      runSig { ExternalAccessible := 'False'; ExternalVisible := 'False'; ExternalWritable := 'False'} : Bool;   // run signal for drive
      errOffDelTime { ExternalAccessible := 'False'; ExternalVisible := 'False'; ExternalWritable := 'False'} : Time := T#1S;   // err off delayed time
      limMin { ExternalAccessible := 'False'; ExternalVisible := 'False'; ExternalWritable := 'False'} : Real;   // minimum limit position (0 = deactivated )
      limMax { ExternalAccessible := 'False'; ExternalVisible := 'False'; ExternalWritable := 'False'} : Real;   // maximum limit position (0 = deactivated )
   END_VAR
   VAR_OUTPUT
      comOk { ExternalAccessible := 'False'; ExternalVisible := 'False'; ExternalWritable := 'False'} : Bool;   // communication ok/active
      ready { ExternalAccessible := 'False'; ExternalVisible := 'False'; ExternalWritable := 'False'} : Bool;   // ready to work
      encAct { ExternalAccessible := 'False'; ExternalVisible := 'False'; ExternalWritable := 'False'} : DInt;   // actual position from counter
      delta { ExternalAccessible := 'False'; ExternalVisible := 'False'; ExternalWritable := 'False'} : Real;   // delta in millimeter
      resetPos { ExternalAccessible := 'False'; ExternalVisible := 'False'; ExternalWritable := 'False'} : Real;   // last reset position for the encoder value (ex. division sensor)
      act { ExternalAccessible := 'False'; ExternalVisible := 'False'; ExternalWritable := 'False'} : Real;   // actual position in millimeter
      sync { ExternalAccessible := 'False'; ExternalVisible := 'False'; ExternalWritable := 'False'} : Bool;   // reset puls (division sensor, or generate with offset)
      err { ExternalAccessible := 'False'; ExternalVisible := 'False'; ExternalWritable := 'False'} : Bool;   // fault
      errCom { ExternalAccessible := 'False'; ExternalVisible := 'False'; ExternalWritable := 'False'} : Bool;   // fault communication
      errRdEnc { ExternalAccessible := 'False'; ExternalVisible := 'False'; ExternalWritable := 'False'} : Bool;   // fault encoder from count module
      errRunCheck { ExternalAccessible := 'False'; ExternalVisible := 'False'; ExternalWritable := 'False'} : Bool;   // fault plausibility check run-signal/encoder-value
      errLim { ExternalAccessible := 'False'; ExternalVisible := 'False'; ExternalWritable := 'False'} : Bool;   // fault position is outside from limits
      errOverFlow { ExternalAccessible := 'False'; ExternalVisible := 'False'; ExternalWritable := 'False'} : Bool;   // fault implausible change in encoder value detected (maybe overflow or underflow)
   END_VAR
   VAR_IN_OUT
      Enc : "TypeEncoder";
   END_VAR
   VAR
      var { ExternalAccessible := 'False'; ExternalVisible := 'False'; ExternalWritable := 'False'; S7_SetPoint := 'True'} : "TypeVar";
      T { ExternalAccessible := 'False'; ExternalVisible := 'False'; ExternalWritable := 'False'; S7_SetPoint := 'True'} : Array[1..3] of IEC_TIMER;
      Rd { ExternalAccessible := 'False'; ExternalVisible := 'False'; ExternalWritable := 'False'} : Struct
         cntBit24 : Bool;   // count value
         stsDI1 : Bool;   // DI1 status
         stsDir : Bool;   // direction
         stsDI0 : Bool;   // DI0 status
         err : Bool;   // fault
         stsDI2 : Bool;   // Tm Count: status DI2
         stsReady : Bool;   // ready
         Wd : Bool;   // watchdog if used isochronous mode
         cntValue2 : Byte;   // count value
         cntValue : Word;   // count value
      END_STRUCT;
      encActOld { ExternalAccessible := 'False'; ExternalVisible := 'False'; ExternalWritable := 'False'} : DInt;
      deltaIncOld { ExternalAccessible := 'False'; ExternalVisible := 'False'; ExternalWritable := 'False'} : DInt;
      actualNoOffset { ExternalAccessible := 'False'; ExternalVisible := 'False'; ExternalWritable := 'False'} : Real;
      errLimMin { ExternalAccessible := 'False'; ExternalVisible := 'False'; ExternalWritable := 'False'} : Bool;
      errLimMax { ExternalAccessible := 'False'; ExternalVisible := 'False'; ExternalWritable := 'False'} : Bool;
   END_VAR
   VAR_TEMP
      tempDelta1 : DInt;
      tempRdRetVal : Int;
      tempErrOverFlow : Bool;
   END_VAR
   VAR_TEMP   // added for the SCL form of the ladder/FBD networks
      _w1 : Bool;
      _w2 : Bool;
   END_VAR
BEGIN

REGION Network 1: exit
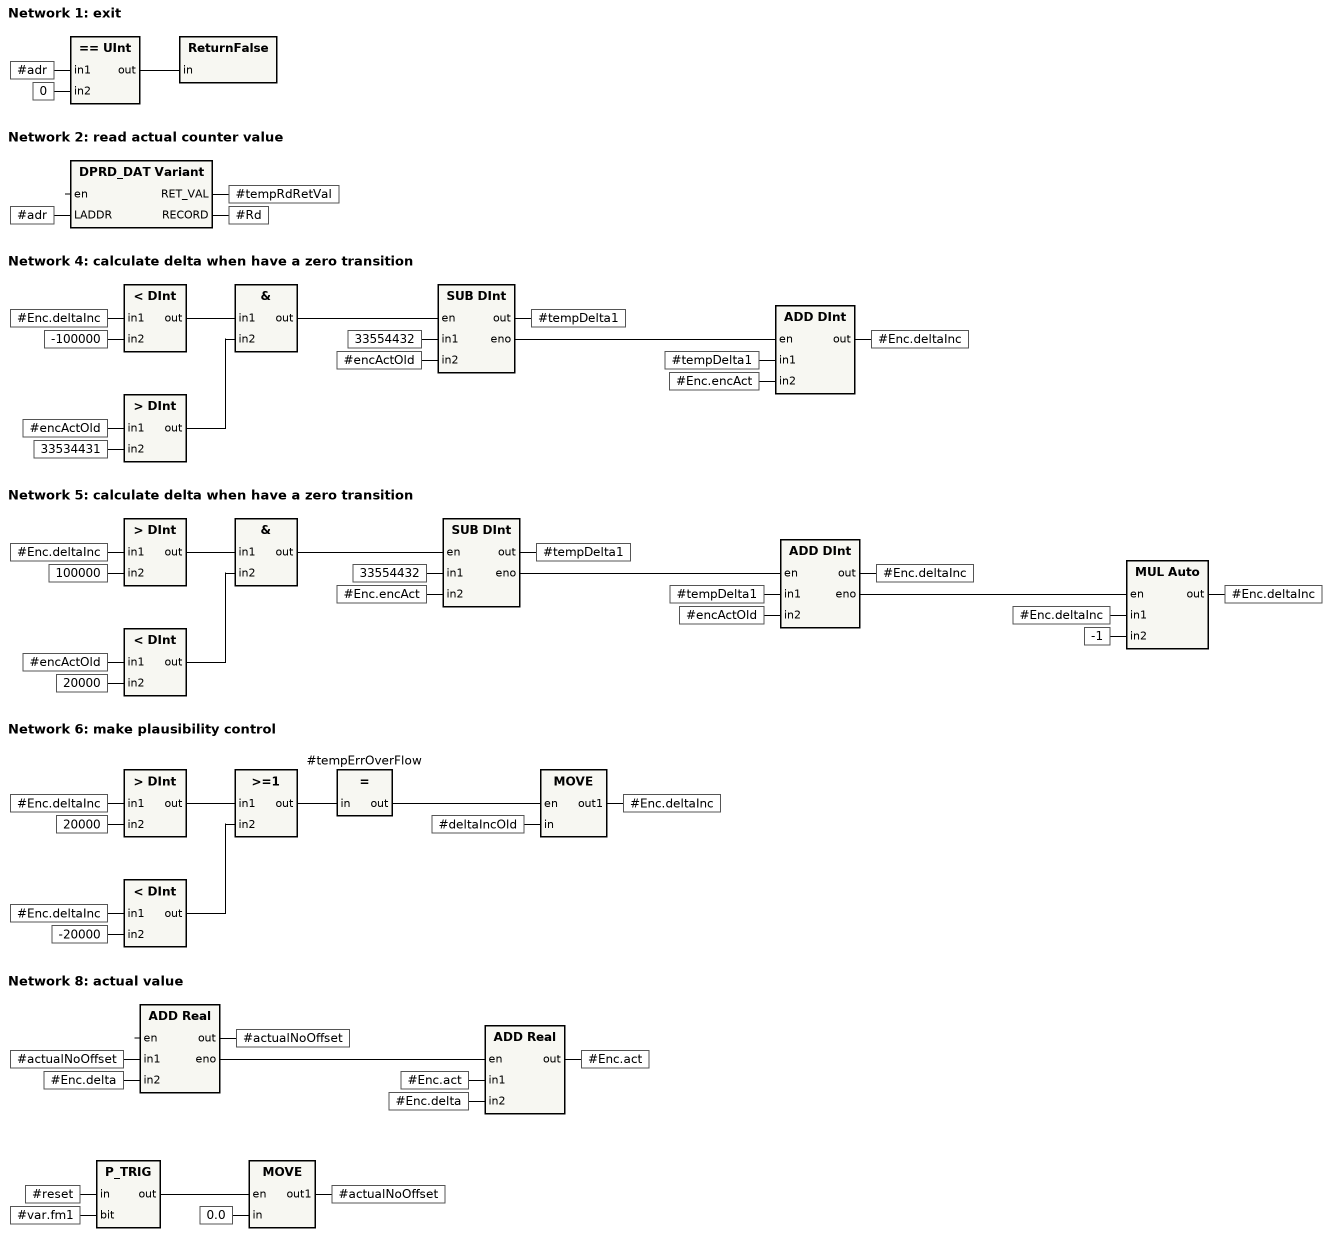
   IF #adr = 0 THEN
       ENO := FALSE;
       RETURN;
   END_IF;
END_REGION

REGION Network 2: read actual counter value
   #tempRdRetVal := DPRD_DAT(LADDR := #adr, RECORD => #Rd);
END_REGION

REGION Network 3 (SCL): read/write values

   #Enc.ready := #Rd.stsReady;
   #Enc.encAct :=  WORD_TO_DWORD(#Rd.cntValue) OR SHL_DWORD(IN:=BYTE_TO_DWORD(#Rd.cntValue2), N:=16);
   #Enc.encAct.%X24 := #Rd.cntBit24;
   #Enc.calOffset := #calOffset;
   #Enc.refPos := #setValue;
   #Enc.limMin := #limMin;
   #Enc.limMax := #limMax;
   #Enc.dirUp := #Rd.stsDir;
   #Enc.dirDn := NOT #Rd.stsDir;

   IF #calGain <> 0.0 THEN
       #Enc.calGain := #calGain;
   ELSE
       #Enc.calGain := 1.0;
   END_IF;

   #Enc.deltaInc := #Enc.encAct - #encActOld;
END_REGION

REGION Network 4: calculate delta when have a zero transition
   // ENO of a box is taken as its EN; it also drops when the box reports an error
   IF (#Enc.deltaInc < (-100000)) AND (#encActOld > 33534431) THEN
       #tempDelta1 := 33554432 - #encActOld;
       #Enc.deltaInc := #tempDelta1 + #Enc.encAct;
   END_IF;
END_REGION

REGION Network 5: calculate delta when have a zero transition
   // ENO of a box is taken as its EN; it also drops when the box reports an error
   IF (#Enc.deltaInc > 100000) AND (#encActOld < 20000) THEN #tempDelta1 := 33554432 - #Enc.encAct; END_IF;
   #_w1 := (#Enc.deltaInc > 100000) AND (#encActOld < 20000);
   IF #_w1 THEN
       #Enc.deltaInc := #tempDelta1 + #encActOld;
       #Enc.deltaInc := #Enc.deltaInc * (-1);
   END_IF;
END_REGION

REGION Network 6: make plausibility control
   #tempErrOverFlow := (#Enc.deltaInc > 20000) OR (#Enc.deltaInc < (-20000));
   IF #tempErrOverFlow THEN #Enc.deltaInc := #deltaIncOld; END_IF;
END_REGION

REGION Network 7 (SCL): increment in mm and actual speed in meter/min
   #Enc.delta := DINT_TO_REAL( #Enc.deltaInc) * #Enc.calGain;
   #Enc.speed := #Enc.speed * 0.9 + (#Enc.delta * 60.0 / "cycle") * 0.1;

   //save old value
   #deltaIncOld := #Enc.deltaInc;
   #encActOld := #Enc.encAct;
END_REGION

REGION Network 8: actual value
   // ENO of a box is taken as its EN; it also drops when the box reports an error
   #actualNoOffset := #actualNoOffset + #Enc.delta;
   #Enc.act := #Enc.act + #Enc.delta;
   #_w1 := #reset AND NOT #var.fm1;   // rising edge
   #var.fm1 := #reset;
   IF #_w1 THEN #actualNoOffset := 0.0; END_IF;
END_REGION

REGION Network 9: virtual reset
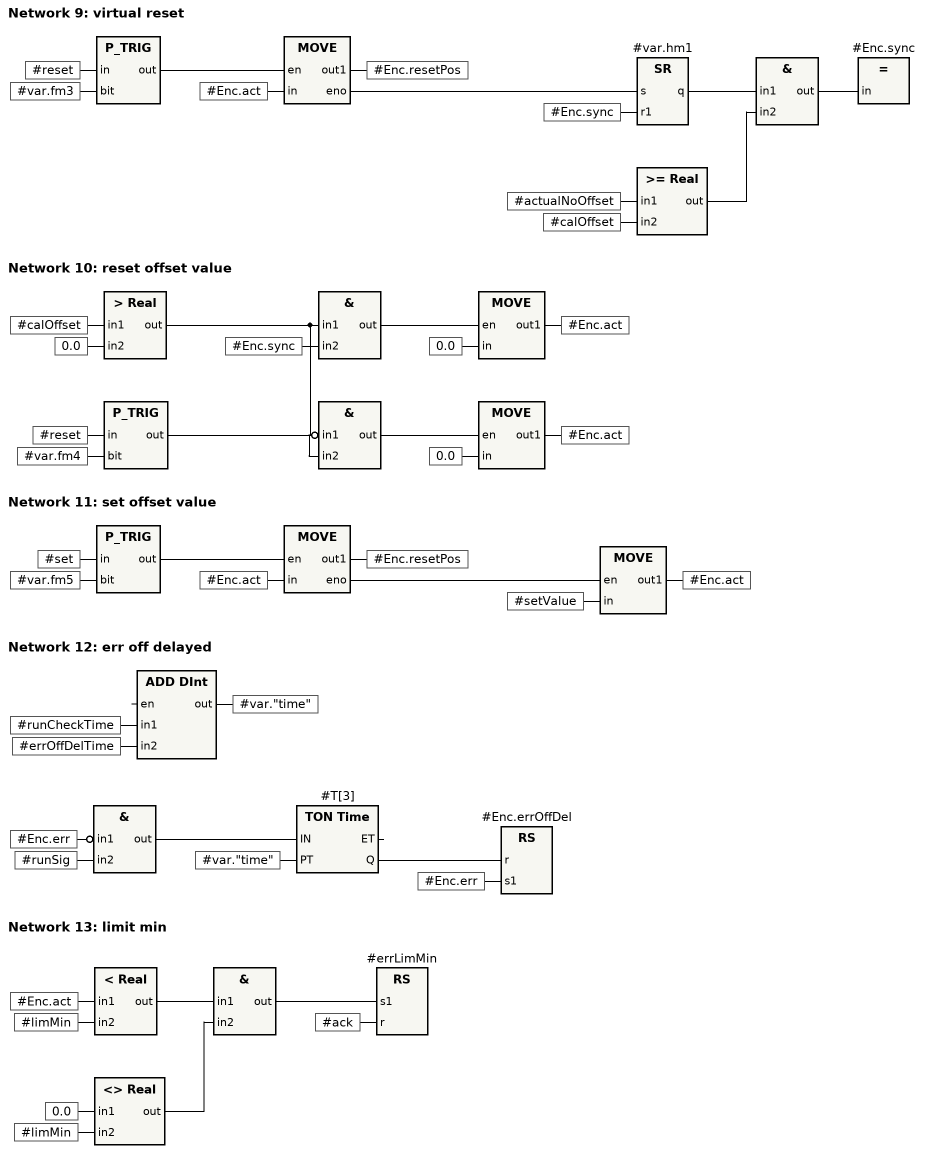
   #_w1 := #reset AND NOT #var.fm3;   // rising edge
   #var.fm3 := #reset;
   IF #_w1 THEN
       #Enc.resetPos := #Enc.act;
       #var.hm1 := TRUE;   // SR flip-flop
   END_IF;
   IF #Enc.sync THEN #var.hm1 := FALSE; END_IF;
   #Enc.sync := #var.hm1 AND (#actualNoOffset >= #calOffset);
END_REGION

REGION Network 10: reset offset value
   #_w1 := #calOffset > 0.0;
   IF #_w1 AND #Enc.sync THEN #Enc.act := 0.0; END_IF;
   #_w2 := #reset AND NOT #var.fm4;   // rising edge
   #var.fm4 := #reset;
   IF NOT #_w1 AND #_w2 THEN #Enc.act := 0.0; END_IF;
END_REGION

REGION Network 11: set offset value
   #_w1 := #set AND NOT #var.fm5;   // rising edge
   #var.fm5 := #set;
   IF #_w1 THEN
       #Enc.resetPos := #Enc.act;
       #Enc.act := #setValue;
   END_IF;
END_REGION

REGION Network 12: err off delayed
   #var."time" := #runCheckTime + #errOffDelTime;
   #T[3].TON(IN := NOT #Enc.err AND #runSig, PT := #var."time");
   IF #T[3].Q THEN
       #Enc.errOffDel := FALSE;   // RS flip-flop
   END_IF;
   IF #Enc.err THEN #Enc.errOffDel := TRUE; END_IF;
END_REGION

REGION Network 13: limit min
   IF #ack THEN
       #errLimMin := FALSE;   // RS flip-flop
   END_IF;
   IF (#Enc.act < #limMin) AND (0.0 <> #limMin) THEN #errLimMin := TRUE; END_IF;
END_REGION

REGION Network 14: limit max
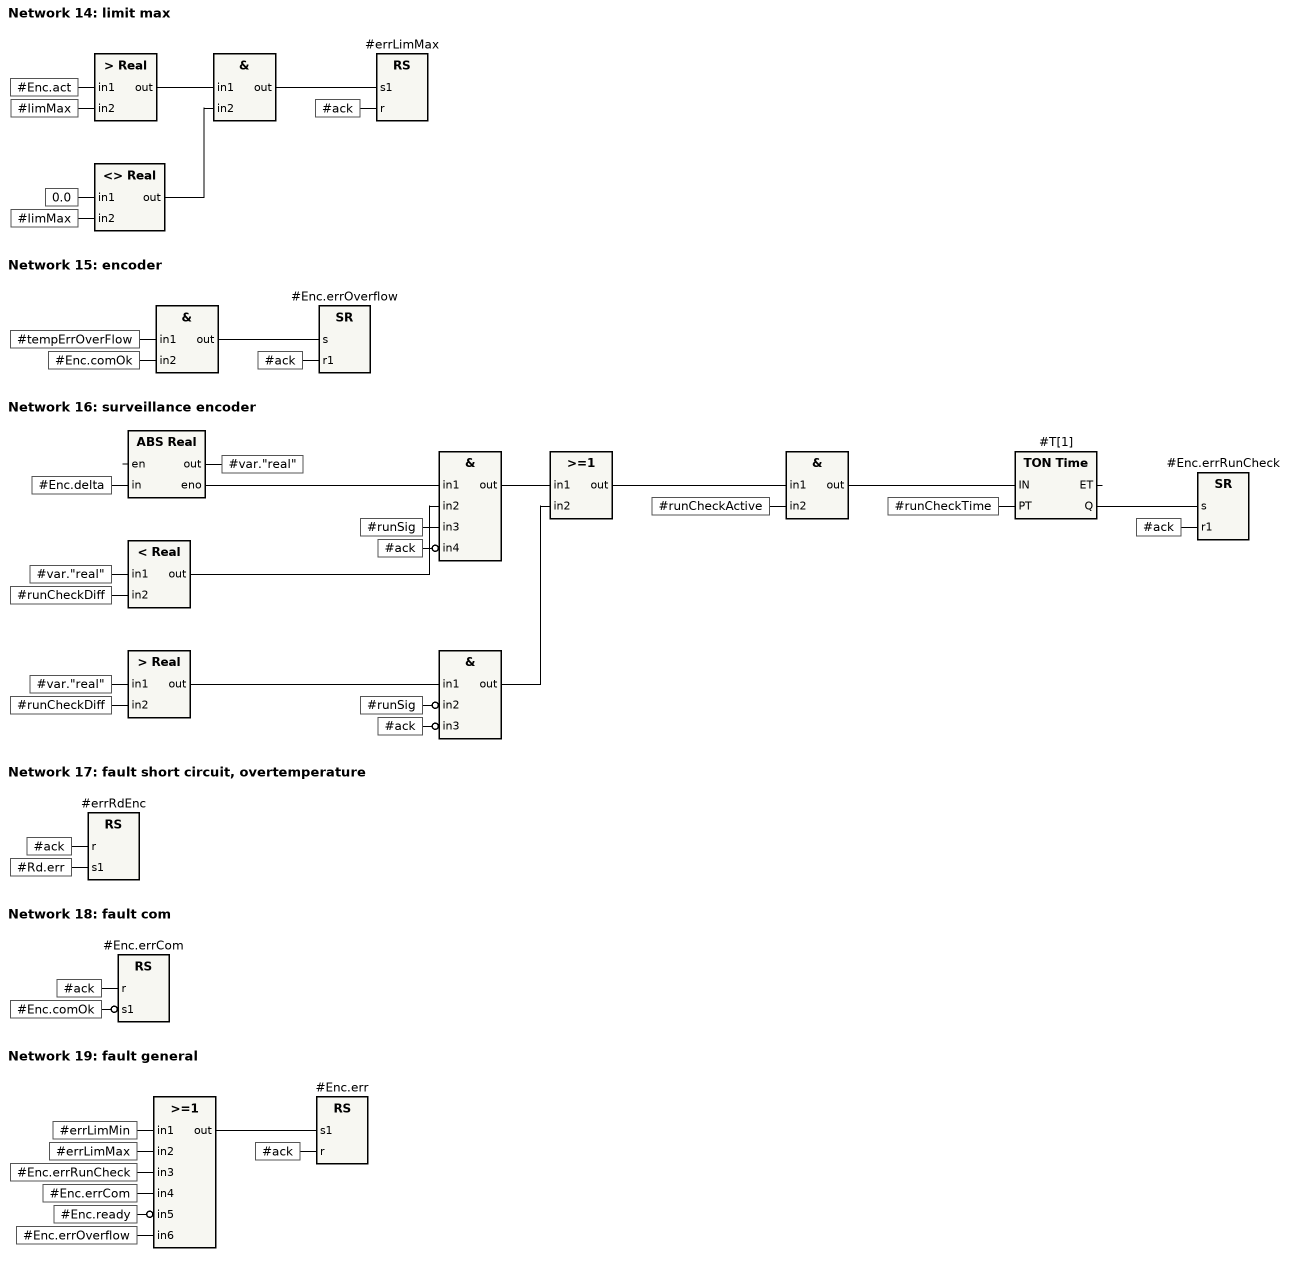
   IF #ack THEN
       #errLimMax := FALSE;   // RS flip-flop
   END_IF;
   IF (#Enc.act > #limMax) AND (0.0 <> #limMax) THEN #errLimMax := TRUE; END_IF;
END_REGION

REGION Network 15: encoder
   IF #tempErrOverFlow AND #Enc.comOk THEN
       #Enc.errOverflow := TRUE;   // SR flip-flop
   END_IF;
   IF #ack THEN #Enc.errOverflow := FALSE; END_IF;
END_REGION

REGION Network 16: surveillance encoder
   #var."real" := ABS(#Enc.delta);
   #T[1].TON(IN := (((#var."real" < #runCheckDiff) AND #runSig AND NOT #ack) OR ((#var."real" > #runCheckDiff) AND NOT #runSig AND NOT #ack)) AND #runCheckActive,
             PT := #runCheckTime);
   IF #T[1].Q THEN
       #Enc.errRunCheck := TRUE;   // SR flip-flop
   END_IF;
   IF #ack THEN #Enc.errRunCheck := FALSE; END_IF;
END_REGION

REGION Network 17: fault short circuit, overtemperature
   IF #ack THEN
       #errRdEnc := FALSE;   // RS flip-flop
   END_IF;
   IF #Rd.err THEN #errRdEnc := TRUE; END_IF;
END_REGION

REGION Network 18: fault com
   IF #ack THEN
       #Enc.errCom := FALSE;   // RS flip-flop
   END_IF;
   IF NOT #Enc.comOk THEN #Enc.errCom := TRUE; END_IF;
END_REGION

REGION Network 19: fault general
   IF #ack THEN
       #Enc.err := FALSE;   // RS flip-flop
   END_IF;
   IF #errLimMin OR #errLimMax OR #Enc.errRunCheck OR #Enc.errCom OR NOT #Enc.ready OR #Enc.errOverflow THEN
       #Enc.err := TRUE;
   END_IF;
END_REGION

REGION Network 20: error number counter [1-50]
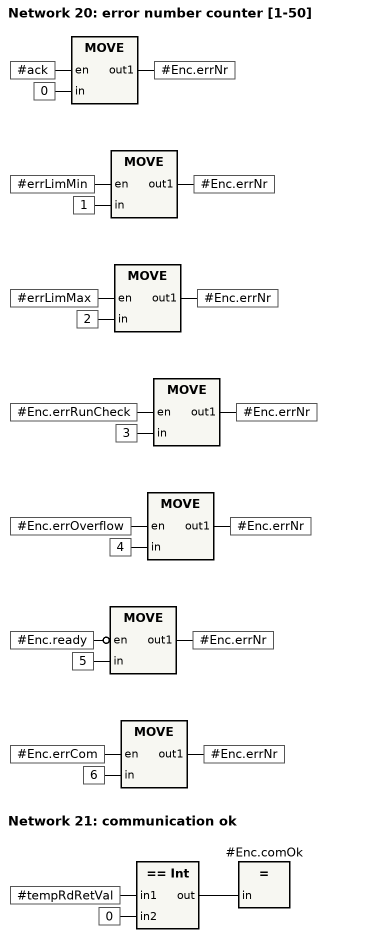
   IF #ack THEN #Enc.errNr := 0; END_IF;
   IF #errLimMin THEN #Enc.errNr := 1; END_IF;
   IF #errLimMax THEN #Enc.errNr := 2; END_IF;
   IF #Enc.errRunCheck THEN #Enc.errNr := 3; END_IF;
   IF #Enc.errOverflow THEN #Enc.errNr := 4; END_IF;
   IF NOT #Enc.ready THEN #Enc.errNr := 5; END_IF;
   IF #Enc.errCom THEN #Enc.errNr := 6; END_IF;
END_REGION

REGION Network 21: communication ok
   #Enc.comOk := #tempRdRetVal = 0;
END_REGION

REGION Network 22 (SCL): write to outputs and encoder data
   #comOk := #Enc.comOk;
   #ready := #Enc.ready;

   #encAct := #Enc.encAct;
   #delta := #Enc.delta;
   #act := #Enc.act ;
   #resetPos := #Enc.resetPos;
   #sync := #Enc.sync;

   #err := #Enc.err;
   #errCom := #Enc.errCom ;
   #errRunCheck := #Enc.errRunCheck ;
   #errLim := #errLimMin OR #errLimMax;
   #errOverFlow := #Enc.errOverflow;

   #Enc.errLim := #errLimMin OR #errLimMax;
   //#Enc.refOk := NOT #Enc.errLim;
END_REGION
END_FUNCTION_BLOCK

FUNCTION_BLOCK "SysSensor"   // FB2040, FBD
TITLE = manage a sensor
{ S7_Optimized_Access := 'TRUE' }
AUTHOR : MiCROTEC
VERSION : 1.5
// -2021.12 : Martin / -2018.12 : Martin
// stored: AutoNumber false, MemoryReserve 100, SetENOAutomatically false
   VAR_INPUT
      errOccIn { ExternalAccessible := 'False'; ExternalVisible := 'False'; ExternalWritable := 'False'} : Bool;   // fault input (sensor signal or a combination of sensors)
      errOccVal { ExternalAccessible := 'False'; ExternalVisible := 'False'; ExternalWritable := 'False'} : Real;   // fault value for fault input
      errFreeIn { ExternalAccessible := 'False'; ExternalVisible := 'False'; ExternalWritable := 'False'} : Bool;   // fault input 2 (sensor signal or a combination of sensors)
      errFreeVal { ExternalAccessible := 'False'; ExternalVisible := 'False'; ExternalWritable := 'False'} : Real;   // fault value for fault input 2
      errCycleIn { ExternalAccessible := 'False'; ExternalVisible := 'False'; ExternalWritable := 'False'} : Bool;   // fault cycle input (this input increment a counter, counter is reset with rise or fallinge edge of sensor )
      errCycleVal { ExternalAccessible := 'False'; ExternalVisible := 'False'; ExternalWritable := 'False'} : Real;   // fault cycle value (if counter exceeds this value then error is set )
      sensor { ExternalAccessible := 'False'; ExternalVisible := 'False'; ExternalWritable := 'False'} : Bool;   // sensor signal
      enable { ExternalAccessible := 'False'; ExternalVisible := 'False'; ExternalWritable := 'False'} : Bool;   // if enable is true than the counter count, ex. run message from conv.
      ack { ExternalAccessible := 'False'; ExternalVisible := 'False'; ExternalWritable := 'False'} : Bool;   // acknowledg faults
      onDelVal { ExternalAccessible := 'False'; ExternalVisible := 'False'; ExternalWritable := 'False'} : Real;   // delayed on value for delayed on
      offDelVal { ExternalAccessible := 'False'; ExternalVisible := 'False'; ExternalWritable := 'False'} : Real;   // delayed off value for delayed off
      occOnVal { ExternalAccessible := 'False'; ExternalVisible := 'False'; ExternalWritable := 'False'} : Real;   // delayed on value for sensor occupied
      occOffVal { ExternalAccessible := 'False'; ExternalVisible := 'False'; ExternalWritable := 'False'} : Real;   // delayed off value for sensor occupied
      cntrVal { ExternalAccessible := 'False'; ExternalVisible := 'False'; ExternalWritable := 'False'} : Real;   // count value per cycle, if absolut encoder than activate "Param.AbsolutEncoder"
      absEnc { ExternalAccessible := 'False'; ExternalVisible := 'False'; ExternalWritable := 'False'} : Bool;   // activate absolut encoder for "countValue"
      reset { ExternalAccessible := 'False'; ExternalVisible := 'False'; ExternalWritable := 'False'} : Bool;   // reset the counter values and also the outputs
   END_VAR
   VAR_OUTPUT
      err { ExternalAccessible := 'False'; ExternalVisible := 'False'; ExternalWritable := 'False'} : Bool;   // Sensor fault , sensor is broken or is dirty
      errOcc { ExternalAccessible := 'False'; ExternalVisible := 'False'; ExternalWritable := 'False'} : Bool;   // Sensor fault , was to long occupied, maybe dirty or misaligned
      errFree { ExternalAccessible := 'False'; ExternalVisible := 'False'; ExternalWritable := 'False'} : Bool;   // Sensor fault , was to long free, maybe dirty or misaligned
      errCycle { ExternalAccessible := 'False'; ExternalVisible := 'False'; ExternalWritable := 'False'} : Bool;   // Sensor fault , plausibility check of cycles, after a certain amount(#errCycleVal) of trigger(#errCycleIn) the sensor had no rising or falling edge
      onDel { ExternalAccessible := 'False'; ExternalVisible := 'False'; ExternalWritable := 'False'} : Bool;   // sensor on delayed
      offDel { ExternalAccessible := 'False'; ExternalVisible := 'False'; ExternalWritable := 'False'} : Bool;   // sensor off delayed
      occ { ExternalAccessible := 'False'; ExternalVisible := 'False'; ExternalWritable := 'False'} : Bool;   // sensor occupied
      onCntr { ExternalAccessible := 'False'; ExternalVisible := 'False'; ExternalWritable := 'False'} : Real;   // counter for on delayed (if sensor is occupied it count, if free than reset)
      offCntr { ExternalAccessible := 'False'; ExternalVisible := 'False'; ExternalWritable := 'False'} : Real;   // counter for off delayed (if sensor is free it count, if occupied than reset)
      occOnCntr { ExternalAccessible := 'False'; ExternalVisible := 'False'; ExternalWritable := 'False'} : Real;   // on counter for occupied (if "occ" is "1" it count, if "0" than reset)
      occOffCntr { ExternalAccessible := 'False'; ExternalVisible := 'False'; ExternalWritable := 'False'} : Real;   // on counter for occupied (if "occ" is "0" it count, if "1" than reset)
   END_VAR
   VAR_IN_OUT
      Sen : "TypeSensor";
   END_VAR
   VAR
      var { ExternalAccessible := 'False'; ExternalVisible := 'False'; ExternalWritable := 'False'} : Struct
         "bool" : Bool;
         "byte" : Byte;
         "word" : Word;
         "dword" : DWord;
         "int" : Int;
         "dint" : DInt;
         "real" : Real;
         s5time : S5Time;
         "time" : Time;
         hm : Array[1..16] of Bool;
         fm : Array[1..16] of Bool;
      END_STRUCT;
      T { ExternalAccessible := 'False'; ExternalVisible := 'False'; ExternalWritable := 'False'} : Array[1..2] of IEC_TIMER;
      cntrValue { ExternalAccessible := 'False'; ExternalVisible := 'False'; ExternalWritable := 'False'} : Real;
      cntrValueOld { ExternalAccessible := 'False'; ExternalVisible := 'False'; ExternalWritable := 'False'} : Real;
      cntrErrOcc { ExternalAccessible := 'False'; ExternalVisible := 'False'; ExternalWritable := 'False'} : Real;   // counter for fault
      cntrErrFree { ExternalAccessible := 'False'; ExternalVisible := 'False'; ExternalWritable := 'False'} : Real;
      cntrErrCycle { ExternalAccessible := 'False'; ExternalVisible := 'False'; ExternalWritable := 'False'} : Real;
   END_VAR
   VAR_TEMP   // added for the SCL form of the ladder/FBD networks
      _w1 : Bool;
      _w2 : Bool;
      _w3 : Bool;
      _w4 : Bool;
   END_VAR
BEGIN

REGION Network 1: counter value value/perCycle or absolut encoder
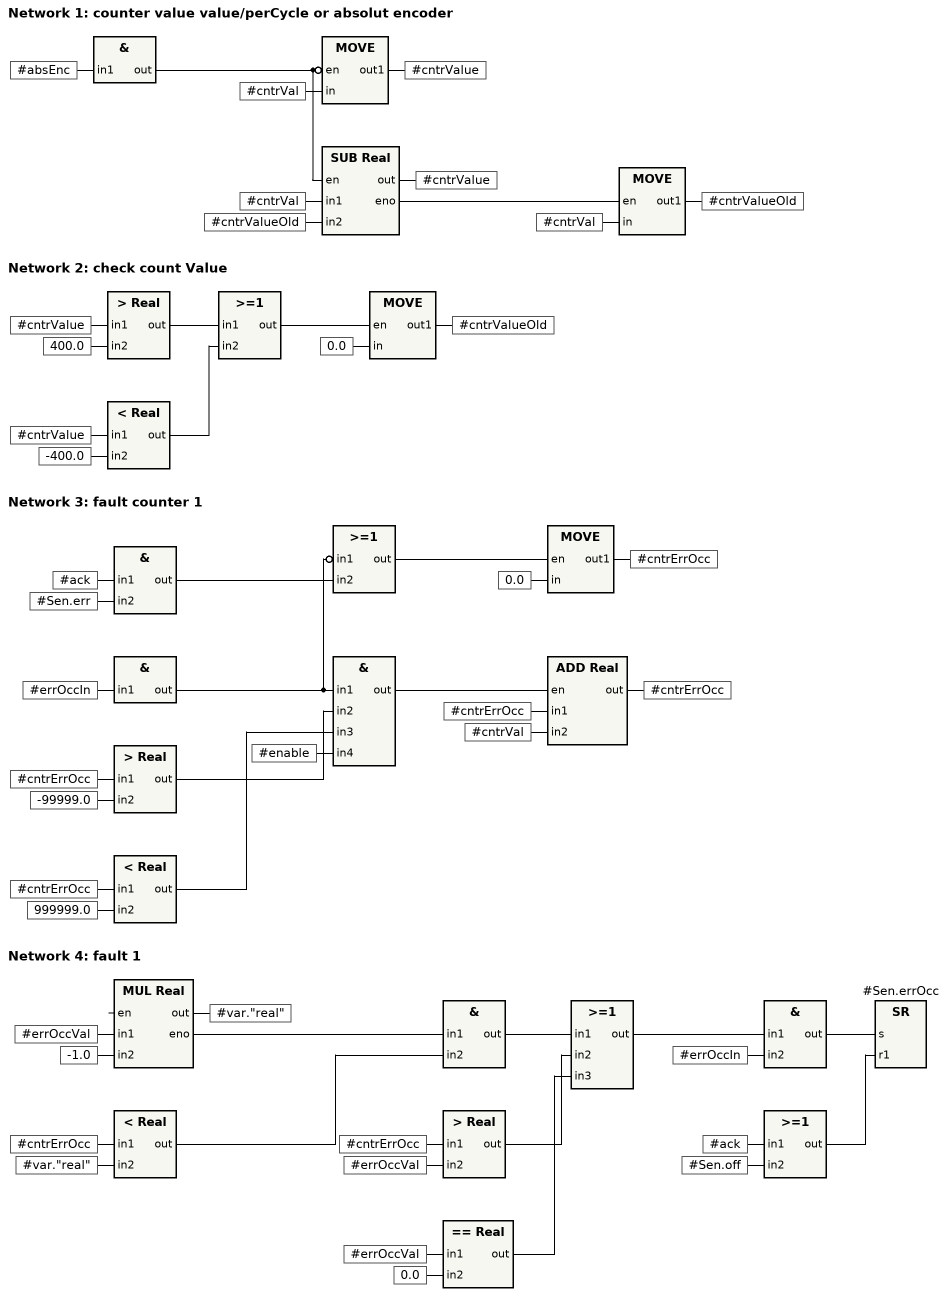
   // ENO of a box is taken as its EN; it also drops when the box reports an error
   IF NOT #absEnc THEN #cntrValue := #cntrVal; END_IF;
   IF #absEnc THEN
       #cntrValue := #cntrVal - #cntrValueOld;
       #cntrValueOld := #cntrVal;
   END_IF;
END_REGION

REGION Network 2: check count Value
   IF (#cntrValue > 400.0) OR (#cntrValue < (-400.0)) THEN #cntrValueOld := 0.0; END_IF;
END_REGION

REGION Network 3: fault counter 1
   IF NOT #errOccIn OR (#ack AND #Sen.err) THEN #cntrErrOcc := 0.0; END_IF;
   IF #errOccIn AND (#cntrErrOcc > (-99999.0)) AND (#cntrErrOcc < 999999.0) AND #enable THEN
       #cntrErrOcc := #cntrErrOcc + #cntrVal;
   END_IF;
END_REGION

REGION Network 4: fault 1
   // ENO of a box is taken as its EN; it also drops when the box reports an error
   #var."real" := #errOccVal * (-1.0);
   IF ((#cntrErrOcc < #var."real") OR (#cntrErrOcc > #errOccVal) OR (#errOccVal = 0.0)) AND #errOccIn THEN
       #Sen.errOcc := TRUE;   // SR flip-flop
   END_IF;
   IF #ack OR #Sen.off THEN #Sen.errOcc := FALSE; END_IF;
END_REGION

REGION Network 5: fault counter 2
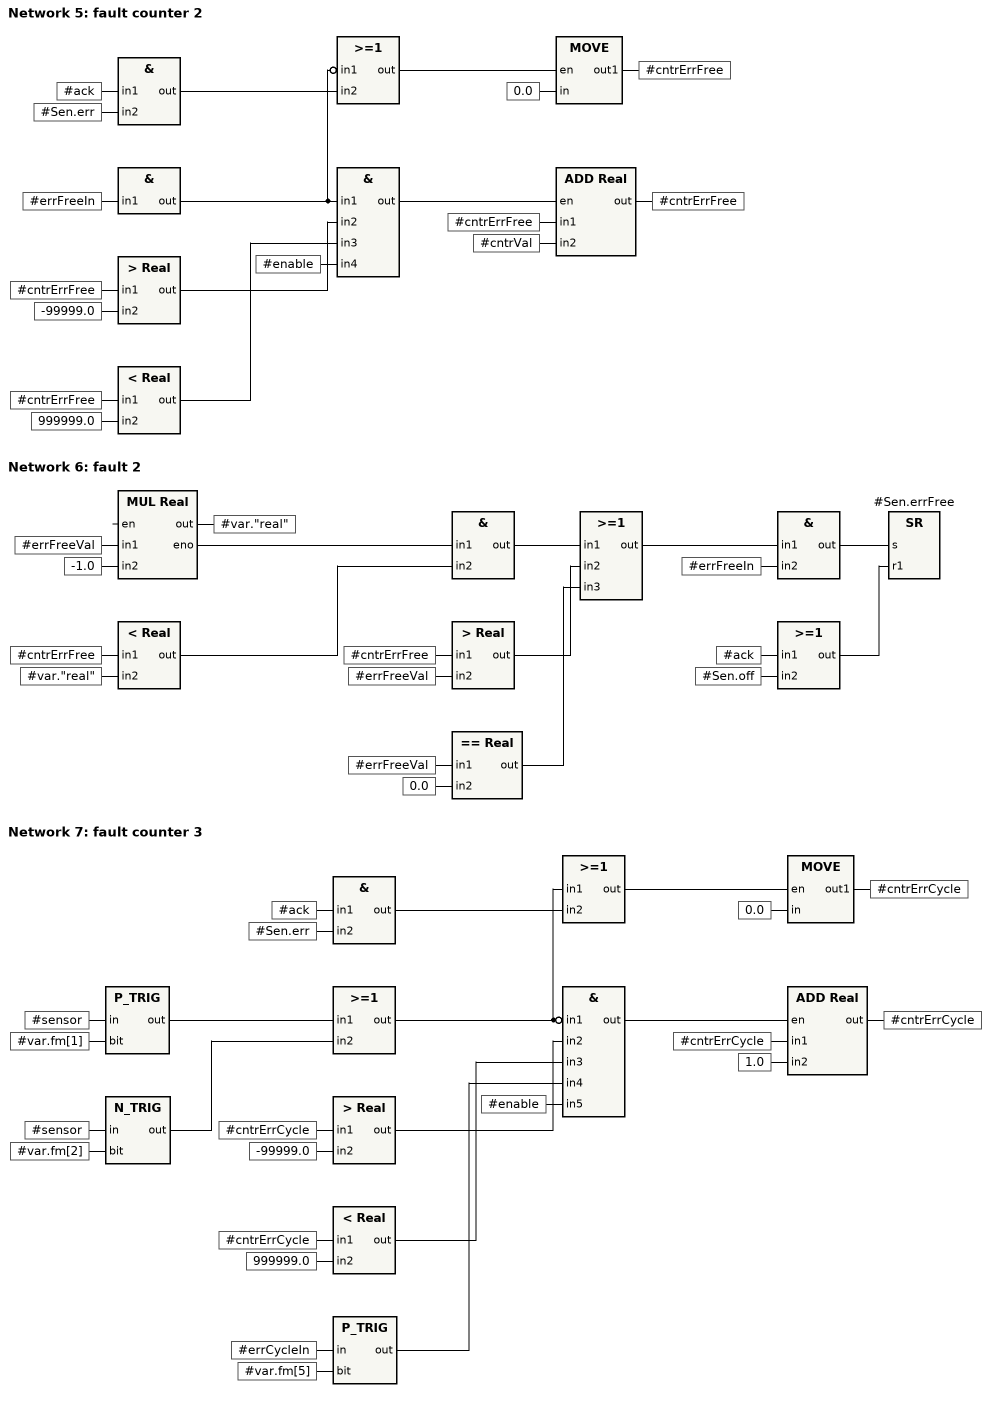
   IF NOT #errFreeIn OR (#ack AND #Sen.err) THEN #cntrErrFree := 0.0; END_IF;
   IF #errFreeIn AND (#cntrErrFree > (-99999.0)) AND (#cntrErrFree < 999999.0) AND #enable THEN
       #cntrErrFree := #cntrErrFree + #cntrVal;
   END_IF;
END_REGION

REGION Network 6: fault 2
   // ENO of a box is taken as its EN; it also drops when the box reports an error
   #var."real" := #errFreeVal * (-1.0);
   IF ((#cntrErrFree < #var."real") OR (#cntrErrFree > #errFreeVal) OR (#errFreeVal = 0.0)) AND #errFreeIn THEN
       #Sen.errFree := TRUE;   // SR flip-flop
   END_IF;
   IF #ack OR #Sen.off THEN #Sen.errFree := FALSE; END_IF;
END_REGION

REGION Network 7: fault counter 3
   #_w1 := #sensor AND NOT #var.fm[1];   // rising edge
   #var.fm[1] := #sensor;
   #_w2 := NOT #sensor AND #var.fm[2];   // falling edge
   #var.fm[2] := #sensor;
   #_w3 := #_w1 OR #_w2;
   IF #_w3 OR (#ack AND #Sen.err) THEN #cntrErrCycle := 0.0; END_IF;
   #_w4 := #errCycleIn AND NOT #var.fm[5];   // rising edge
   #var.fm[5] := #errCycleIn;
   IF NOT #_w3 AND (#cntrErrCycle > (-99999.0)) AND (#cntrErrCycle < 999999.0) AND #_w4 AND #enable THEN
       #cntrErrCycle := #cntrErrCycle + 1.0;
   END_IF;
END_REGION

REGION Network 8: fault 3
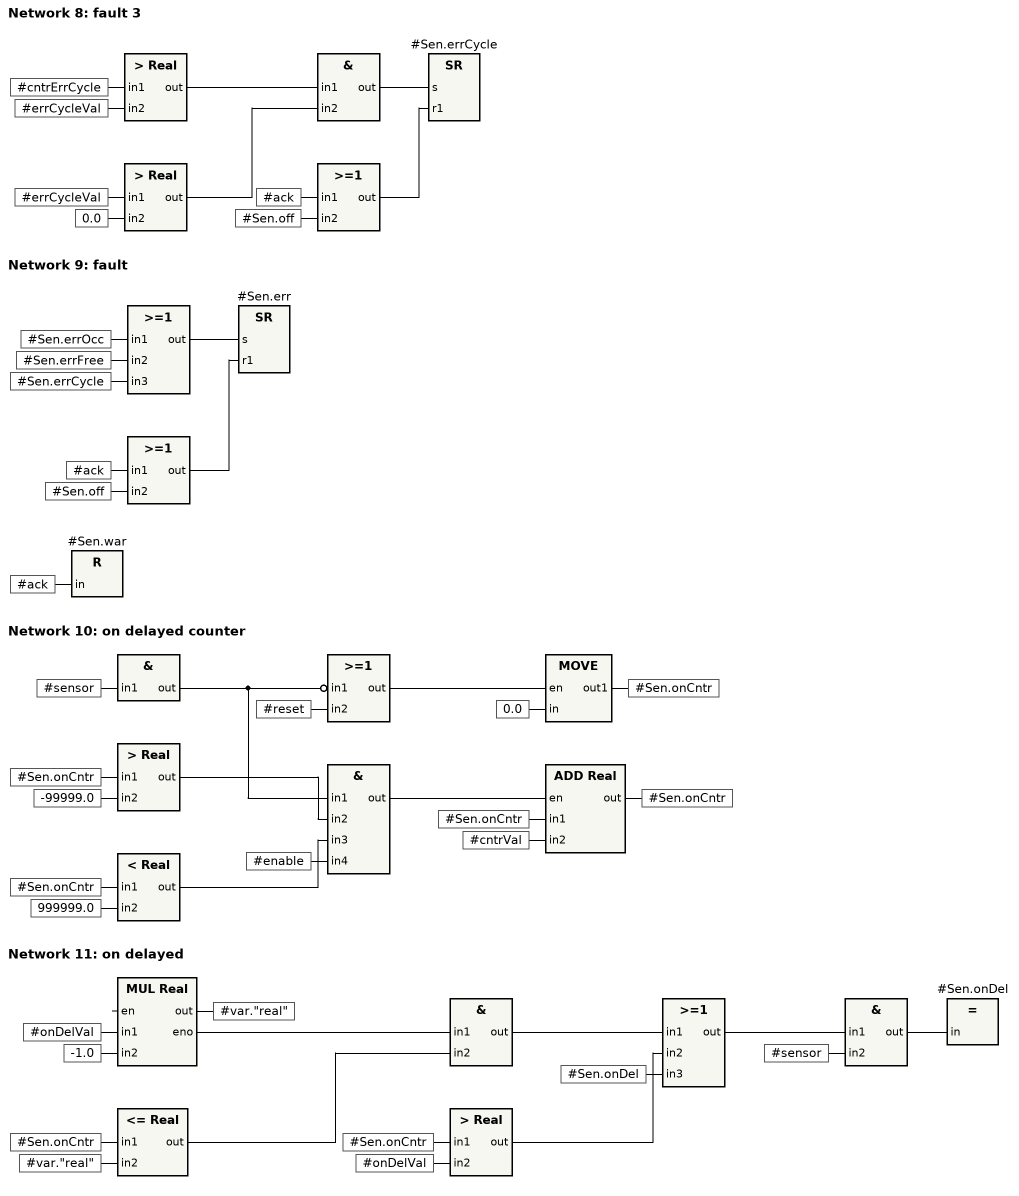
   IF (#cntrErrCycle > #errCycleVal) AND (#errCycleVal > 0.0) THEN
       #Sen.errCycle := TRUE;   // SR flip-flop
   END_IF;
   IF #ack OR #Sen.off THEN #Sen.errCycle := FALSE; END_IF;
END_REGION

REGION Network 9: fault
   IF #Sen.errOcc OR #Sen.errFree OR #Sen.errCycle THEN
       #Sen.err := TRUE;   // SR flip-flop
   END_IF;
   IF #ack OR #Sen.off THEN #Sen.err := FALSE; END_IF;
   IF #ack THEN #Sen.war := FALSE; END_IF;
END_REGION

REGION Network 10: on delayed counter
   IF NOT #sensor OR #reset THEN #Sen.onCntr := 0.0; END_IF;
   IF #sensor AND (#Sen.onCntr > (-99999.0)) AND (#Sen.onCntr < 999999.0) AND #enable THEN
       #Sen.onCntr := #Sen.onCntr + #cntrVal;
   END_IF;
END_REGION

REGION Network 11: on delayed
   // ENO of a box is taken as its EN; it also drops when the box reports an error
   #var."real" := #onDelVal * (-1.0);
   #Sen.onDel := ((#Sen.onCntr <= #var."real") OR (#Sen.onCntr > #onDelVal) OR #Sen.onDel) AND #sensor;
END_REGION

REGION Network 12: off delayed counter
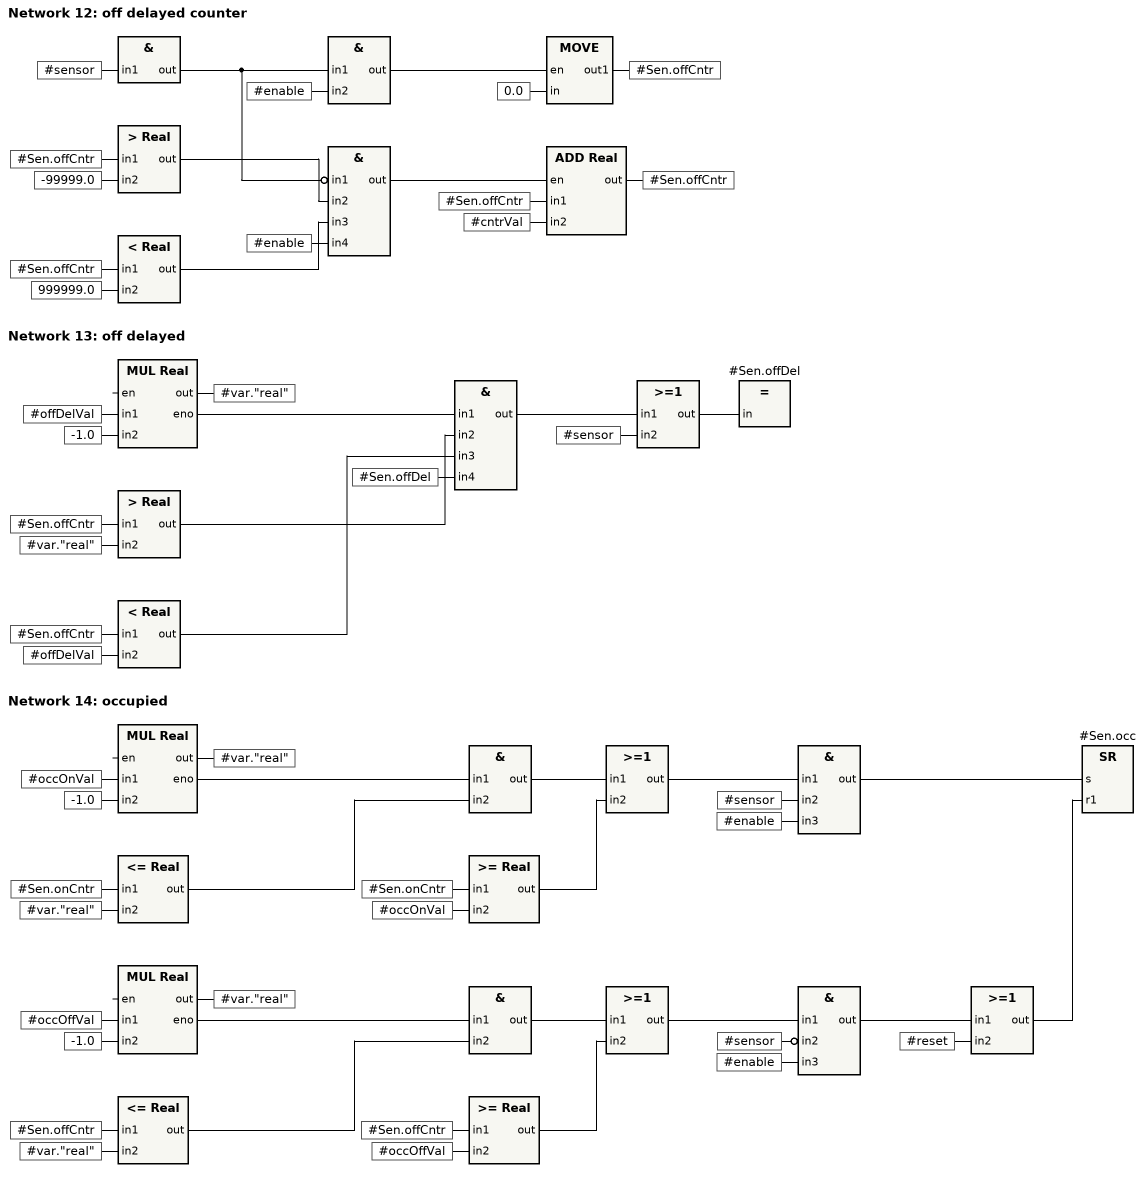
   IF #sensor AND #enable THEN #Sen.offCntr := 0.0; END_IF;
   IF NOT #sensor AND (#Sen.offCntr > (-99999.0)) AND (#Sen.offCntr < 999999.0) AND #enable THEN
       #Sen.offCntr := #Sen.offCntr + #cntrVal;
   END_IF;
END_REGION

REGION Network 13: off delayed
   // ENO of a box is taken as its EN; it also drops when the box reports an error
   #var."real" := #offDelVal * (-1.0);
   #Sen.offDel := ((#Sen.offCntr > #var."real") AND (#Sen.offCntr < #offDelVal) AND #Sen.offDel) OR #sensor;
END_REGION

REGION Network 14: occupied
   // ENO of a box is taken as its EN; it also drops when the box reports an error
   #var."real" := #occOnVal * (-1.0);
   #_w1 := ((#Sen.onCntr <= #var."real") OR (#Sen.onCntr >= #occOnVal)) AND #sensor AND #enable;
   #var."real" := #occOffVal * (-1.0);
   IF #_w1 THEN
       #Sen.occ := TRUE;   // SR flip-flop
   END_IF;
   IF (((#Sen.offCntr <= #var."real") OR (#Sen.offCntr >= #occOffVal)) AND NOT #sensor AND #enable) OR #reset THEN
       #Sen.occ := FALSE;
   END_IF;
END_REGION

REGION Network 15: positive / negative edge
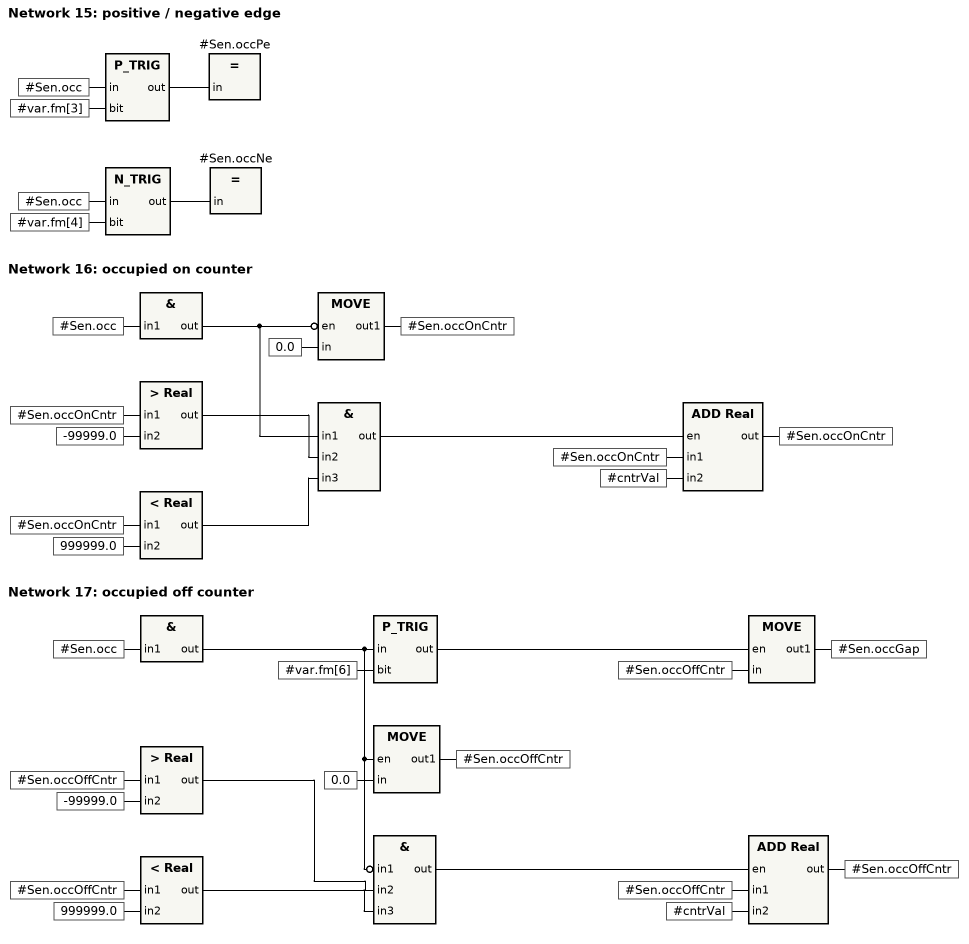
   #_w1 := #Sen.occ AND NOT #var.fm[3];   // rising edge
   #var.fm[3] := #Sen.occ;
   #Sen.occPe := #_w1;
   #_w2 := NOT #Sen.occ AND #var.fm[4];   // falling edge
   #var.fm[4] := #Sen.occ;
   #Sen.occNe := #_w2;
END_REGION

REGION Network 16: occupied on counter
   IF NOT #Sen.occ THEN #Sen.occOnCntr := 0.0; END_IF;
   IF #Sen.occ AND (#Sen.occOnCntr > (-99999.0)) AND (#Sen.occOnCntr < 999999.0) THEN
       #Sen.occOnCntr := #Sen.occOnCntr + #cntrVal;
   END_IF;
END_REGION

REGION Network 17: occupied off counter
   #_w1 := #Sen.occ AND NOT #var.fm[6];   // rising edge
   #var.fm[6] := #Sen.occ;
   IF #_w1 THEN #Sen.occGap := #Sen.occOffCntr; END_IF;
   IF #Sen.occ THEN #Sen.occOffCntr := 0.0; END_IF;
   IF NOT #Sen.occ AND (#Sen.occOffCntr > (-99999.0)) AND (#Sen.occOffCntr < 999999.0) THEN
       #Sen.occOffCntr := #Sen.occOffCntr + #cntrVal;
   END_IF;
END_REGION

REGION Network 18 (SCL): write outputs
      #err := #Sen.err;
       #errOcc := #Sen.errOcc;
       #errFree := #Sen.errFree;
       #errCycle := #Sen.errCycle;
       #onDel :=  #Sen.onDel;
       #offDel :=  #Sen.offDel;
       #occ := #Sen.occ;
       #onCntr :=  #Sen.onCntr;
       #offCntr := #Sen.offCntr;
       #occOnCntr :=    #Sen.occOnCntr ;
       #occOffCntr :=  #Sen.occOffCntr;

       #Sen.sen := #sensor;
END_REGION
END_FUNCTION_BLOCK

FUNCTION_BLOCK "SysWenglorP3PC301"   // FB4011, FBD
{ S7_Optimized_Access := 'TRUE' }
// stored: AutoNumber false, MemoryReserve 100, SetENOAutomatically false
   VAR_INPUT
      adrHW { ExternalAccessible := 'False'; ExternalVisible := 'False'; ExternalWritable := 'False'} : HW_IO;   // I/O adress HW
      adr { ExternalAccessible := 'False'; ExternalVisible := 'False'; ExternalWritable := 'False'} : Int;   // I/O adress
      slot { ExternalAccessible := 'False'; ExternalVisible := 'False'; ExternalWritable := 'False'} : Int;   // slot of io link module 1..4
      ack { ExternalAccessible := 'False'; ExternalVisible := 'False'; ExternalWritable := 'False'} : Bool;   // acknowledge
      laserOff { ExternalAccessible := 'False'; ExternalVisible := 'False'; ExternalWritable := 'False'} : Bool;   // Laser off
      findMe { ExternalAccessible := 'False'; ExternalVisible := 'False'; ExternalWritable := 'False'} : Bool;   // Find me, flash sensor led
      teachA1 { ExternalAccessible := 'False'; ExternalVisible := 'False'; ExternalWritable := 'False'} : Bool;   // teach A1
      teachA2 { ExternalAccessible := 'False'; ExternalVisible := 'False'; ExternalWritable := 'False'} : Bool;   // teach A2
      startConfig { ExternalAccessible := 'False'; ExternalVisible := 'False'; ExternalWritable := 'False'} : Bool;
   END_VAR
   VAR_OUTPUT
      Measure { ExternalAccessible := 'False'; ExternalVisible := 'False'; ExternalWritable := 'False'} : Real;   // Actual measured value [mm] (-1= Read error)
      Scale { ExternalAccessible := 'False'; ExternalVisible := 'False'; ExternalWritable := 'False'} : Real;   // Scale -6 = µm
      ComOk { ExternalAccessible := 'False'; ExternalVisible := 'False'; ExternalWritable := 'False'} : Bool;   // communication ok
      ConfigOk { ExternalAccessible := 'False'; ExternalVisible := 'False'; ExternalWritable := 'False'} : Bool;   // configuration ok
      MeasureOk { ExternalAccessible := 'False'; ExternalVisible := 'False'; ExternalWritable := 'False'} : Bool;   // measuring ok
      Err { ExternalAccessible := 'False'; ExternalVisible := 'False'; ExternalWritable := 'False'} : Bool;   // Signal sensor error (1= Error)
      Warn { ExternalAccessible := 'False'; ExternalVisible := 'False'; ExternalWritable := 'False'} : Bool;   // Signal sensorwarning (1= Dirty)
      A1 { ExternalAccessible := 'False'; ExternalVisible := 'False'; ExternalWritable := 'False'} : Bool;   // Signal output 1 (1= Occ)
      A2 { ExternalAccessible := 'False'; ExternalVisible := 'False'; ExternalWritable := 'False'} : Bool;   // Signal output 2 (1= Occ)
   END_VAR
   VAR_IN_OUT
      param : "TypeIOLinkParamArray";
   END_VAR
   VAR
      var { ExternalAccessible := 'False'; ExternalVisible := 'False'; ExternalWritable := 'False'} : Struct
         "bool" : Bool;
         "byte" : Byte;
         "word" : Word;
         "dword" : DWord;
         "int" : Int;
         "dint" : DInt;
         "real" : Real;
         s5time : S5Time;
         "time" : Time;
         hm : Array[1..50] of Bool;
         fm : Array[1..50] of Bool;
      END_STRUCT;
      Rd { ExternalAccessible := 'False'; ExternalVisible := 'False'; ExternalWritable := 'False'} : "TypeWenglorP3PC301Rd";
      Sd { ExternalAccessible := 'False'; ExternalVisible := 'False'; ExternalWritable := 'False'} : "TypeWenglorP3PC301Sd";
      Data { ExternalAccessible := 'False'; ExternalVisible := 'False'; ExternalWritable := 'False'} : Struct
         Measure : Real;
         Scale : Real;
         ComOk : Bool;
         ConfigOk : Bool;
         MeasureOk : Bool;
         A1 : Bool;
         A2 : Bool;
         Warn : Bool;
         Err : Bool;
         ErrCom : Bool;
         ErrSensor : Bool;
         ErrConfig : Bool;
         WarnSensor : Bool;
      END_STRUCT;
      device { ExternalAccessible := 'False'; ExternalVisible := 'False'; ExternalWritable := 'False'} : "LIOLink_Device";
      statRecord { ExternalAccessible := 'False'; ExternalVisible := 'False'; ExternalWritable := 'False'} : Array[0..231] of Byte;
      cfgData { ExternalAccessible := 'False'; ExternalVisible := 'False'; ExternalWritable := 'False'} : Struct
         Index : Int;
         Subindex : Int;
         Len : Int;
         Value : "TypeIOLinkParamData";
      END_STRUCT;
      cfg { ExternalAccessible := 'False'; ExternalVisible := 'False'; ExternalWritable := 'False'} : Struct
         "Step" : Int;
         Done : Bool;
         Active : Bool;
         Err : Bool;
         Restart : Bool;
      END_STRUCT;
      T1 { ExternalAccessible := 'False'; ExternalVisible := 'False'; ExternalWritable := 'False'} : TON_TIME;
      cnt_i { ExternalAccessible := 'False'; ExternalVisible := 'False'; ExternalWritable := 'False'} : Int;
      cnt_y { ExternalAccessible := 'False'; ExternalVisible := 'False'; ExternalWritable := 'False'} : Int;
      cnt_x { ExternalAccessible := 'False'; ExternalVisible := 'False'; ExternalWritable := 'False'} : Int;
   END_VAR
   VAR_TEMP
      t_Data1 : DWord;
      t_Data2 : Byte;
      t_Data3 : Byte;
      t_ENO : Bool;
      t_Output : Byte;
   END_VAR
BEGIN

REGION Network 1 (SCL): info
   (*    
       Serie:          Wenglor P3PCxxx    
       Type:           Wenglor P3PC301
       Range:          60..660mm
       Vendor ID:      87
       Device ID:      4134746
       Input:          6 Byte
       Output:         1 Byte

       Autor:          Alexander Kiebacher
       Datum:          05/2024
       Änderung:       05/2024
       Version:        1.0
       Lizenz:         Microtec

       Revisionen:     V1.0    
   *)
END_REGION

REGION Network 2 (SCL): read data

   #t_Data1 := PEEK_DWORD(area := 16#1, dbNumber := 0, byteOffset := #adr, ENO => #t_ENO);
   #t_Data2 := PEEK_BYTE(area := 16#1, dbNumber := 0, byteOffset := #adr + 4, ENO => #t_ENO);
   #t_Data3 := PEEK_BYTE(area := 16#1, dbNumber := 0, byteOffset := #adr + 5, ENO => #t_ENO);
   ENO := #t_ENO;
END_REGION

REGION Network 3 (SCL): read data - copy data
   // #Data.Scale := WORD_TO_SINT(SHR(IN := #t_Data2 AND 16#FF00, N := 8));
   // 
   // 0x80000008 –2147483640 Objekt zu nah
   // 0x7FFFFFF8 2147483640 Objekt zu weit
   // 0x7FFFFFFC 2147483644 Kein Signal

   IF ENO THEN

       #Rd.Measure := DWORD_TO_DINT(#t_Data1);
       #Rd.Scale := BYTE_TO_SINT(#t_Data2);
       #Rd.SCC1 := #t_Data3.%X0;
       #Rd.SCC2 := #t_Data3.%X1;
       #Rd.Err := #t_Data3.%X2;
       #Rd.Warn := #t_Data3.%X3;
       #Rd.Warn1 := #t_Data3.%X4;
       #Rd.Warn2 := #t_Data3.%X5;
       #Rd.Warn3 := #t_Data3.%X6;
       #Rd.Warn4 := #t_Data3.%X7;

       // check communication
       #Data.MeasureOk := false;
       IF #Rd.Measure <> 0 THEN
           #Data.ComOk := true;
       ELSE
           #Data.ComOk := false;
       END_IF;

       IF #Rd.Measure = 2147483644 THEN        // no measurement data
           #Data.Measure := -1.0;
       ELSIF #Rd.Measure <= -2147483640 THEN   // out of measuring range (-)
           #Data.Measure := -1.0;
       ELSIF #Rd.Measure >= 2147483640 THEN    // out of measuring range (+)
           #Data.Measure := -1.0;
       ELSIF #Data.ComOk THEN
           #Data.Measure := DINT_TO_REAL(#Rd.Measure) / 1000.0 ;
           #Data.MeasureOk := true;
       END_IF;

       #Data.Scale := SINT_TO_REAL(#Rd.Scale);
       #Data.A1 := #Rd.SCC1;
       #Data.A2 := #Rd.SCC2;

   ELSE
       #Data.Measure := -1.0;
       #Data.Scale := 0.0;
       #Data.A1 := false;
       #Data.A2 := false;
       #Data.ComOk := false;

   END_IF;
END_REGION

REGION Network 5: reset fault / warning
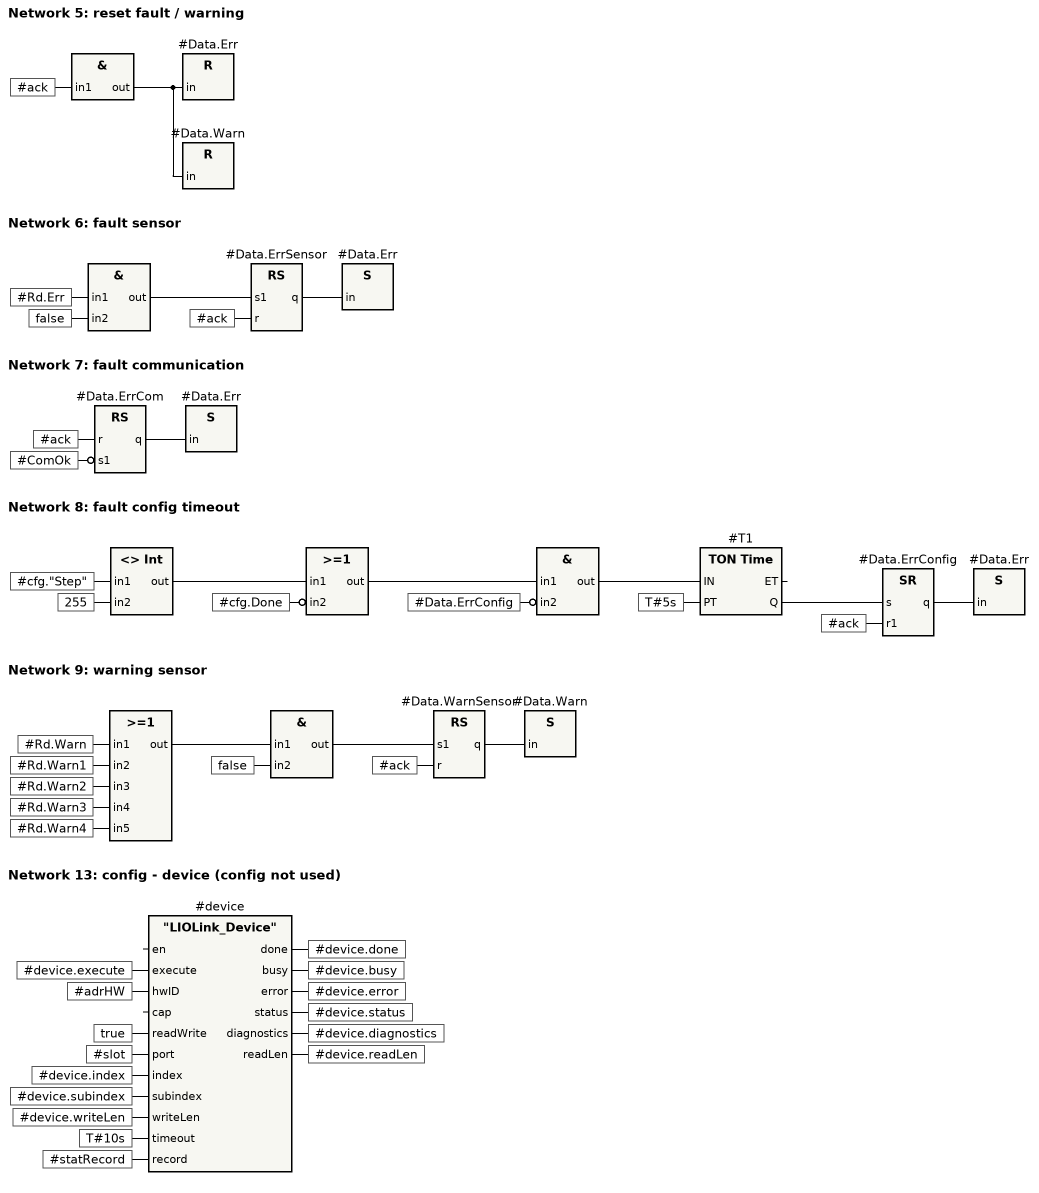
   IF #ack THEN
       #Data.Err := FALSE;
       #Data.Warn := FALSE;
   END_IF;
END_REGION

REGION Network 6: fault sensor
   IF #ack THEN
       #Data.ErrSensor := FALSE;   // RS flip-flop
   END_IF;
   IF #Rd.Err AND false THEN #Data.ErrSensor := TRUE; END_IF;
   IF #Data.ErrSensor THEN #Data.Err := TRUE; END_IF;
END_REGION

REGION Network 7: fault communication
   IF #ack THEN
       #Data.ErrCom := FALSE;   // RS flip-flop
   END_IF;
   IF NOT #ComOk THEN #Data.ErrCom := TRUE; END_IF;
   IF #Data.ErrCom THEN #Data.Err := TRUE; END_IF;
END_REGION

REGION Network 8: fault config timeout
   #T1(IN := ((#cfg."Step" <> 255) OR NOT #cfg.Done) AND NOT #Data.ErrConfig, PT := T#5s);   // TON
   IF #T1.Q THEN
       #Data.ErrConfig := TRUE;   // SR flip-flop
   END_IF;
   IF #ack THEN #Data.ErrConfig := FALSE; END_IF;
   IF #Data.ErrConfig THEN #Data.Err := TRUE; END_IF;
END_REGION

REGION Network 9: warning sensor
   IF #ack THEN
       #Data.WarnSensor := FALSE;   // RS flip-flop
   END_IF;
   IF (#Rd.Warn OR #Rd.Warn1 OR #Rd.Warn2 OR #Rd.Warn3 OR #Rd.Warn4) AND false THEN
       #Data.WarnSensor := TRUE;
   END_IF;
   IF #Data.WarnSensor THEN #Data.Warn := TRUE; END_IF;
END_REGION

REGION Network 10 (SCL): send data - copy data

   #Sd.LaserOff := #laserOff;
   #Sd.Localization := #findMe;
   #Sd.SCC1TeachIn := #teachA1;
   #Sd.SCC2TeachIn := #teachA2;

   #t_Output.%X0 := #Sd.LaserOff;
   #t_Output.%X1 := #Sd.Localization;
   #t_Output.%X2 := false;
   #t_Output.%X3 := #Sd.SCC1TeachIn;
   #t_Output.%X4 := #Sd.SCC1TeachIn;
   #t_Output.%X5 := false;
   #t_Output.%X6 := false;
   #t_Output.%X7 := false;
END_REGION

REGION Network 11 (SCL): send data

   POKE(area := 16#82, dbNumber := 0, byteOffset := #adr, value := #t_Output);
END_REGION

REGION Network 13: config - device (config not used)
   #device(execute := #device.execute,   // "LIOLink_Device"
           hwID := #adrHW,
           readWrite := true,
           port := #slot,
           index := #device.index,
           subindex := #device.subindex,
           writeLen := #device.writeLen,
           timeout := T#10s,
           record := #statRecord,
           done => #device.done,
           busy => #device.busy,
           error => #device.error,
           status => #device.status,
           diagnostics => #device.diagnostics,
           readLen => #device.readLen);
END_REGION

REGION Network 14 (SCL): config - device (config not used)
   (* Invalid *)

   IF (#cfg.Step <= 0 OR #cfg.Step > 255 OR #Data.ErrConfig) THEN
       #cfg.Done := false;
       #cfg.Err := true;
       #cfg.Step := 1;
       #device.execute := false;
   END_IF;

   CASE #cfg.Step OF
       1:  (* Not configured or config request *)
           IF (NOT #cfg.Done OR #cfg.Restart) AND NOT #Data.ErrConfig THEN
               #cfg.Done := false;
               #cfg.Restart := false;
               #cfg.Err := true;
               #cfg.Step := 20;
               #cnt_i := 0;
               #device.execute := false;
           END_IF;

   (* Setup correct operation mode *)        
       20: (* Start config  *)

           #cfgData.Index := #param.Param[#cnt_i].Index;
           #cfgData.Subindex := #param.Param[#cnt_i].Subindex;
           #cfgData.Len := #param.Param[#cnt_i].Len;

           FOR #cnt_y := 0 TO (#cfgData.Len - 1) BY 1 DO
               #cfgData.Value.data[#cnt_y] := #param.Param[#cnt_i].Value.data[#cnt_y];
           END_FOR;

           #device.index := #cfgData.Index ;
           #device.subindex := #cfgData.Subindex ;
           #device.writeLen := #cfgData.Len;
           FOR #cnt_x := 0 TO (#cfgData.Len - 1) BY 1 DO
               #statRecord[#cnt_x] := #cfgData.Value.data[#cnt_x];
           END_FOR;

           #device.execute := false;
           #cfg.Step := 21;

       21: (* Start request *)
           #device.execute := true;
           #cfg.Step := 22;

       22: (*Wait for execution *)
           IF #device.done THEN
               #device.execute := false;
               IF #param.Param[#cnt_i + 1].Len <> 0 THEN
                   #cnt_i := #cnt_i + 1;
                   #cfg.Step := 20;
               ELSE
                   #cfg.Step := 255;
               END_IF;

           END_IF;
           IF #device.error THEN
               #device.execute := false;
               #cfg.Step := 20;
           END_IF;

   (* Setup done *)
       255:
           #cfg.Done := true;
           #cfg.Err := false;

           IF #cfg.Done AND #startConfig THEN
               #cfg.Done := false;
               #cfg.Err := true;
               #cfg.Step := 1;
               #device.execute := false;
               #Data.ErrConfig := false;
           END_IF;

   END_CASE;

   #cfg.Active := #cfg.Step > 10 AND #cfg.Step <255;

   #Data.ConfigOk := #cfg.Done;

   IF TRUE THEN

       #Data.ConfigOk := TRUE;
       #cfg.Done := TRUE;
       #cfg.Step := 255;

   END_IF;
END_REGION

REGION Network 15 (SCL): write outputs

   #Measure := #Data.Measure;
   #Scale := #Data.Scale;
   #ComOk := #Data.ComOk;
   #ConfigOk := #Data.ConfigOk;
   #MeasureOk := #Data.MeasureOk;
   #Err := #Data.Err;
   #Warn := #Data.Warn;
   #A1 := #Data.A1;
   #A2 := #Data.A2;
END_REGION
END_FUNCTION_BLOCK

FUNCTION_BLOCK "AdjScanner"   // FB510, FBD
{ S7_Optimized_Access := 'TRUE' }
// stored: AutoNumber false, MemoryReserve 100, SetENOAutomatically false
   VAR
      Var { ExternalAccessible := 'False'; ExternalVisible := 'False'; ExternalWritable := 'False'} : "TypeVar";
      Cmd { ExternalAccessible := 'False'; ExternalVisible := 'False'; ExternalWritable := 'False'} : "TypeCmd";
      SIO { ExternalAccessible := 'False'; ExternalVisible := 'False'; ExternalWritable := 'False'} : "SysBaluffBUS007F";
      Pos { ExternalAccessible := 'False'; ExternalVisible := 'False'; ExternalWritable := 'False'} : "SysPos";
      "M" { ExternalAccessible := 'False'; ExternalVisible := 'False'; ExternalWritable := 'False'} : "SysMotor";
      TAreaOn { ExternalAccessible := 'False'; ExternalVisible := 'False'; ExternalWritable := 'False'} : TON_TIME;
      TAutoOn { ExternalAccessible := 'False'; ExternalVisible := 'False'; ExternalWritable := 'False'} : TON_TIME;
      TAutoTarPosManOn { ExternalAccessible := 'False'; ExternalVisible := 'False'; ExternalWritable := 'False'} : TON_TIME;
      TPosRestart { ExternalAccessible := 'False'; ExternalVisible := 'False'; ExternalWritable := 'False'} : TON_TIME;
      tarOld { ExternalAccessible := 'False'; ExternalVisible := 'False'; ExternalWritable := 'False'} : DInt;
      autoTarPosMan { ExternalAccessible := 'False'; ExternalVisible := 'False'; ExternalWritable := 'False'} : Bool;
      refTarPos { ExternalAccessible := 'False'; ExternalVisible := 'False'; ExternalWritable := 'False'} : DInt;
      posRestart { ExternalAccessible := 'False'; ExternalVisible := 'False'; ExternalWritable := 'False'} : Bool;
      posOk { ExternalAccessible := 'False'; ExternalVisible := 'False'; ExternalWritable := 'False'} : Bool;
      posRegActive { ExternalAccessible := 'False'; ExternalVisible := 'False'; ExternalWritable := 'False'} : Bool;
   END_VAR
   VAR_TEMP
      CtrlPc : Struct
         ackErr : Bool;
         manModeActive : Bool;
         manP : Bool;
         manM : Bool;
         manRefRun : Bool;
      END_STRUCT;
      refPosDiff : DInt;
      areaDelayOn : Bool;
      offsetZeroPoint : Real;
      TarTolMin : Real;
      TarTolMax : Real;
      PosOkTolMin : Real;
      PosOkTolMax : Real;
      tolerance : Real;
      regPoint : Real;
   END_VAR
BEGIN

REGION Network 1 (SCL): calibration value from pc
   "ComSd".Data.Scanner.SetCalibratePosOk := FALSE;

   IF "ComRd".Data.Scanner.SetCalibratePos THEN

       IF "G".Cfg.modeBoardPassing = 3 THEN
           "Enc"."8B1.B".refPos := 0;
       ELSIF "G".Cfg.modeBoardPassing = 2 THEN
           "Enc"."8B1.B".refPos := (DINT_TO_REAL("ComRd".Data.Scanner.TargetPos) / 10.0) * -1.0;
       ELSE
           "Enc"."8B1.B".refPos := DINT_TO_REAL("ComRd".Data.Scanner.TargetPos) / 10.0;
       END_IF;
       "ComSd".Data.Scanner.SetCalibratePosOk := TRUE;
       "Enc"."8B1.B".ref := TRUE;
   END_IF;
END_REGION

REGION Network 2 (SCL): standardisation batch
   (* 
   if standardisation batch is active then the scanner status display should be off
   *)
   IF "ComRd".Data.Scanner.CalibratePos = -1 THEN
       "G".Batch.stdActive := TRUE;
   ELSE
       "G".Batch.stdActive := FALSE;
   END_IF;
END_REGION

REGION Network 3 (SCL): offset scanner
   (* 
   used with left AND right alignement to avoid the problem that a
   camera cannot position because is in mecanical limit switch
   ex.: right camera cannot reach position because is on minimum limit switch,
   so we move the scanner with an offset of 20 mm  more to the right side
   *)
   "Enc"."8B1.B".offset := DINT_TO_REAL(LIMIT_DINT(MN := -50, IN := "ComRd".Data.Scanner.RefPosToBoard, MX := 50));
END_REGION

REGION Network 4 (SCL): target position
   IF "G".comOk THEN
       #Cmd.target := DINT_TO_REAL("ComRd".Data.Scanner.TargetPos) / 10.0;
   END_IF;

   IF "G".Cfg.modeBoardPassing = 3 THEN
       #Cmd.target := 0.0;
   END_IF;

   IF #autoTarPosMan THEN
       #Cmd.target := DINT_TO_REAL("ComRd".Data.Scanner.TargetPos) / 10.0;
   END_IF;

   IF "G".Cfg.modeBoardPassing = 2 THEN
       #Cmd.target := #Cmd.target * -1.0 ;
   END_IF;

   "Ref".adjScannerTar :=  #Cmd.target + "Enc"."8B1.B".offset;
END_REGION

REGION Network 5 (SCL): data from pc
   IF NOT "G".errComPc THEN
       #CtrlPc.manModeActive := "ComRd".Data.Scanner.ManModeActive;
       #CtrlPc.manRefRun := "ComRd".Data.Scanner.ManRefRun;
       IF "G".Cfg.modeBoardPassing = 2 THEN
           #CtrlPc.manP := "ComRd".Data.Scanner.ManMinus;
           #CtrlPc.manM := "ComRd".Data.Scanner.ManPlus;
       ELSE
           #CtrlPc.manP := "ComRd".Data.Scanner.ManPlus;
           #CtrlPc.manM := "ComRd".Data.Scanner.ManMinus;
       END_IF;
   ELSE
       #CtrlPc.manModeActive := TRUE;
       #CtrlPc.manP := FALSE;
       #CtrlPc.manM := FALSE;
       #CtrlPc.manRefRun := FALSE;
   END_IF;
   #CtrlPc.ackErr := "G".ack;
END_REGION

REGION Network 6: off
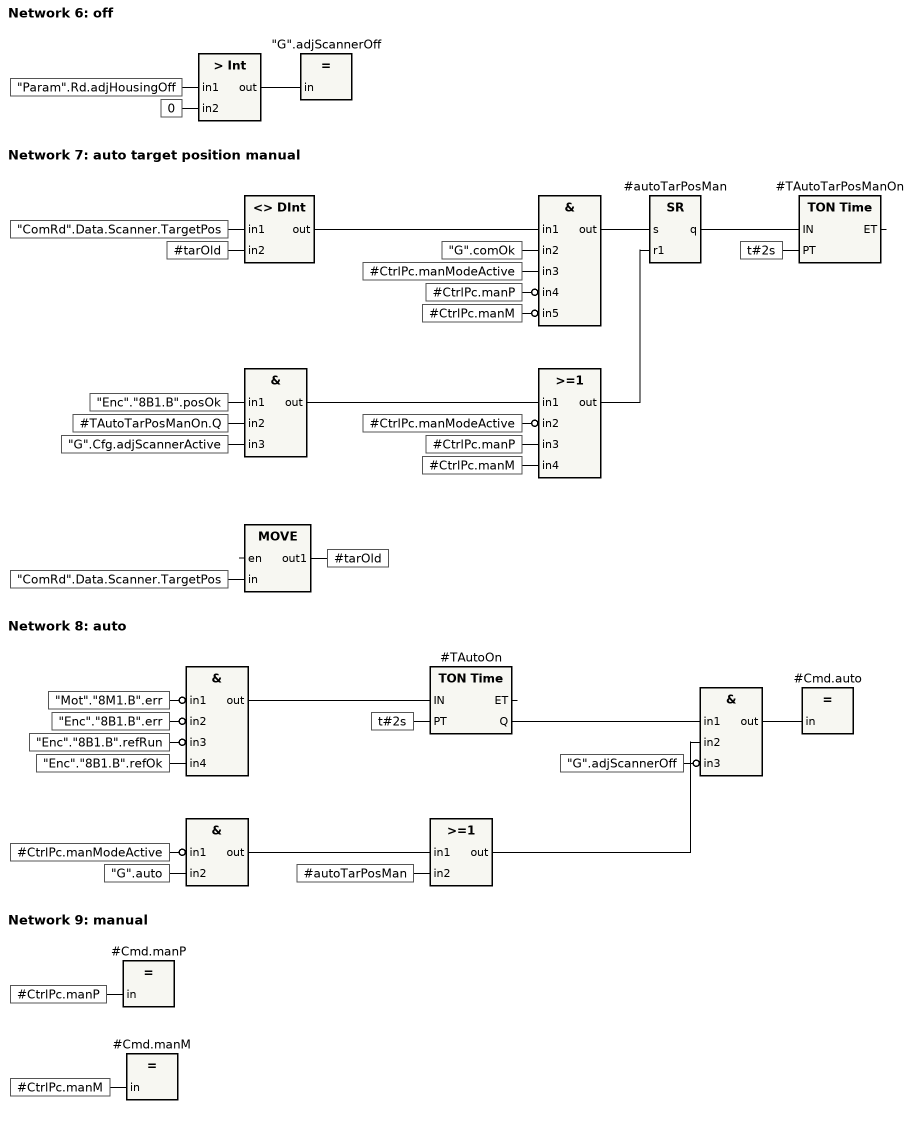
   "G".adjScannerOff := "Param".Rd.adjHousingOff > 0;
END_REGION

REGION Network 7: auto target position manual
   IF ("ComRd".Data.Scanner.TargetPos <> #tarOld) AND "G".comOk AND #CtrlPc.manModeActive AND NOT #CtrlPc.manP AND NOT #CtrlPc.manM THEN
       #autoTarPosMan := TRUE;   // SR flip-flop
   END_IF;
   IF ("Enc"."8B1.B".posOk AND #TAutoTarPosManOn.Q AND "G".Cfg.adjScannerActive) OR NOT #CtrlPc.manModeActive OR #CtrlPc.manP OR #CtrlPc.manM THEN
       #autoTarPosMan := FALSE;
   END_IF;
   #TAutoTarPosManOn(IN := #autoTarPosMan, PT := t#2s);   // TON
   #tarOld := "ComRd".Data.Scanner.TargetPos;
END_REGION

REGION Network 8: auto
   #TAutoOn(IN := NOT "Mot"."8M1.B".err AND NOT "Enc"."8B1.B".err AND NOT "Enc"."8B1.B".refRun AND "Enc"."8B1.B".refOk,   // TON
            PT := t#2s);
   #Cmd.auto := #TAutoOn.Q AND ((NOT #CtrlPc.manModeActive AND "G".auto) OR #autoTarPosMan) AND NOT "G".adjScannerOff;
END_REGION

REGION Network 9: manual
   #Cmd.manP := #CtrlPc.manP;
   #Cmd.manM := #CtrlPc.manM;
END_REGION

REGION Network 10 (SCL): calibration value
   "Enc"."8B1.B".calGain := 0.1;

   "Enc"."8B1.B".minPos := -500.0;
   "Enc"."8B1.B".maxPos := 500.0;

   "Enc"."8B1.B".limMin := "Enc"."8B1.B".minPos - 5.0;
   "Enc"."8B1.B".limMax := "Enc"."8B1.B".maxPos + 5.0;

   "Enc"."8B1.B".tarMinPos := "Enc"."8B1.B".minPos + 0.0;
   "Enc"."8B1.B".tarMaxPos := "Enc"."8B1.B".maxPos - 0.0;

   #offsetZeroPoint := -117.3;
END_REGION

REGION Network 12: sensor IO-Link adjustment scannerhousing
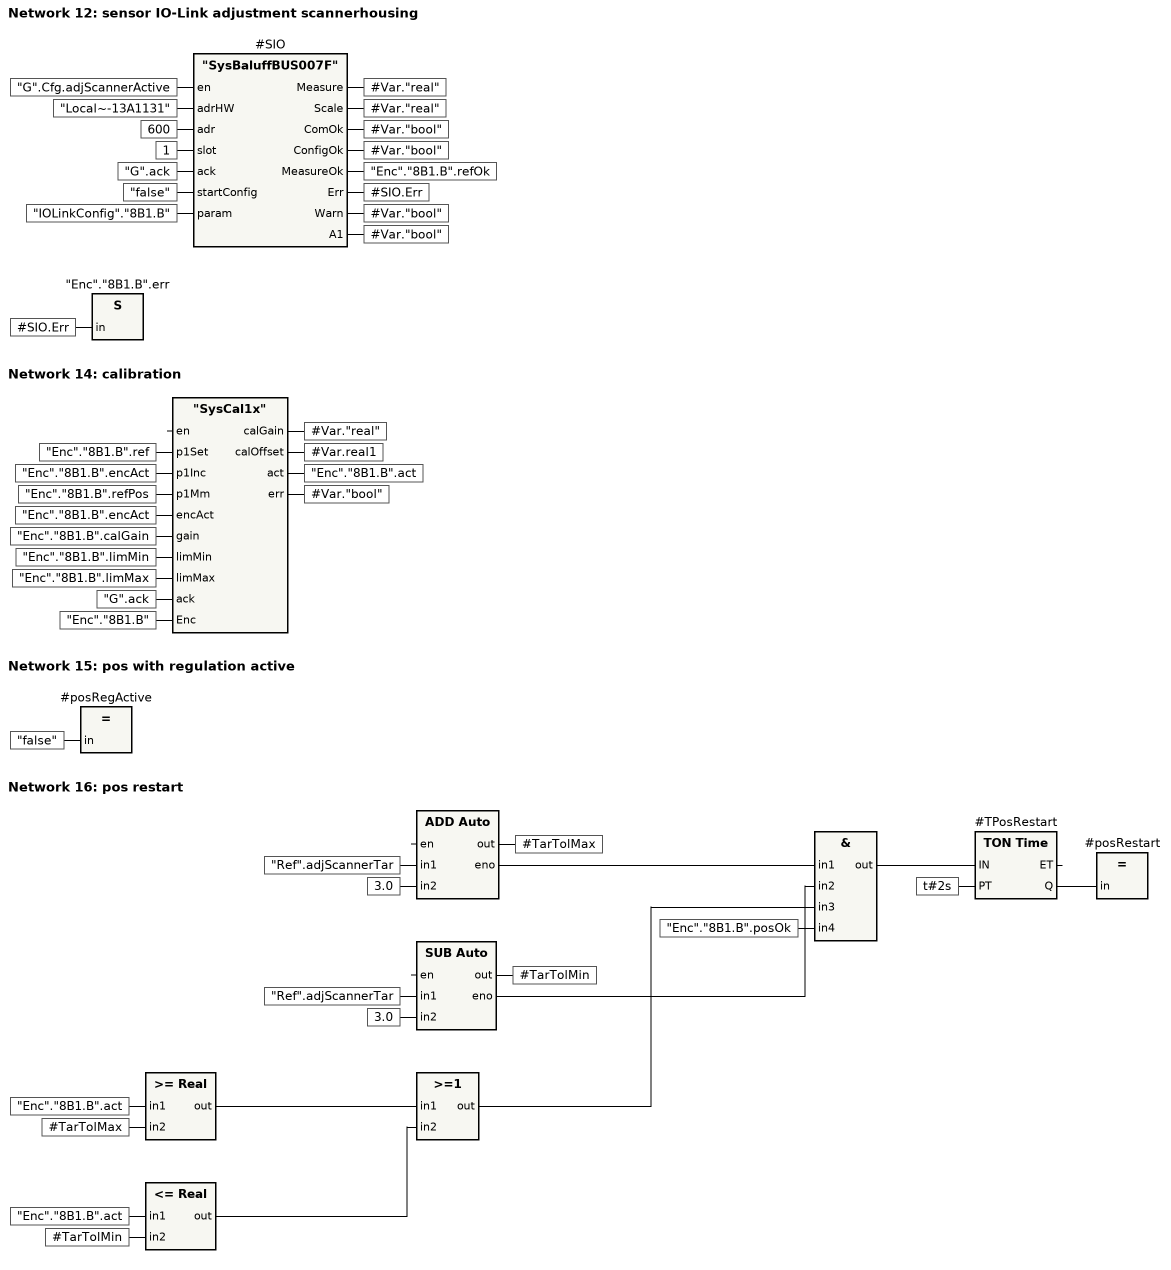
   IF "G".Cfg.adjScannerActive THEN
       #SIO(adrHW := "Local~-13A1131",   // "SysBaluffBUS007F"
            adr := 600,
            slot := 1,
            ack := "G".ack,
            startConfig := "false",
            param := "IOLinkConfig"."8B1.B",
            Measure => #Var."real",
            Scale => #Var."real",
            ComOk => #Var."bool",
            ConfigOk => #Var."bool",
            MeasureOk => "Enc"."8B1.B".refOk,
            Err => #SIO.Err,
            Warn => #Var."bool",
            A1 => #Var."bool");
   END_IF;
   IF #SIO.Err THEN "Enc"."8B1.B".err := TRUE; END_IF;
END_REGION

REGION Network 13 (SCL): sensor IO-Link adjustment scannerhousing - copy data
   "Enc"."8B1.B".encAct := REAL_TO_DINT((#SIO.Measure + #offsetZeroPoint) * 10.0);
END_REGION

REGION Network 14: calibration
   "SysCal1x"(p1Set := "Enc"."8B1.B".ref,
              p1Inc := "Enc"."8B1.B".encAct,
              p1Mm := "Enc"."8B1.B".refPos,
              encAct := "Enc"."8B1.B".encAct,
              gain := "Enc"."8B1.B".calGain,
              limMin := "Enc"."8B1.B".limMin,
              limMax := "Enc"."8B1.B".limMax,
              ack := "G".ack,
              Enc := "Enc"."8B1.B",
              calGain => #Var."real",
              calOffset => #Var.real1,
              act => "Enc"."8B1.B".act,
              err => #Var."bool");
END_REGION

REGION Network 15: pos with regulation active
   #posRegActive := "false";
END_REGION

REGION Network 16: pos restart
   #TarTolMax := "Ref".adjScannerTar + 3.0;
   #TarTolMin := "Ref".adjScannerTar - 3.0;
   #TPosRestart(IN := (("Enc"."8B1.B".act >= #TarTolMax) OR ("Enc"."8B1.B".act <= #TarTolMin)) AND "Enc"."8B1.B".posOk,   // TON
                PT := t#2s);
   #posRestart := #TPosRestart.Q;
END_REGION

REGION Network 17: pos param
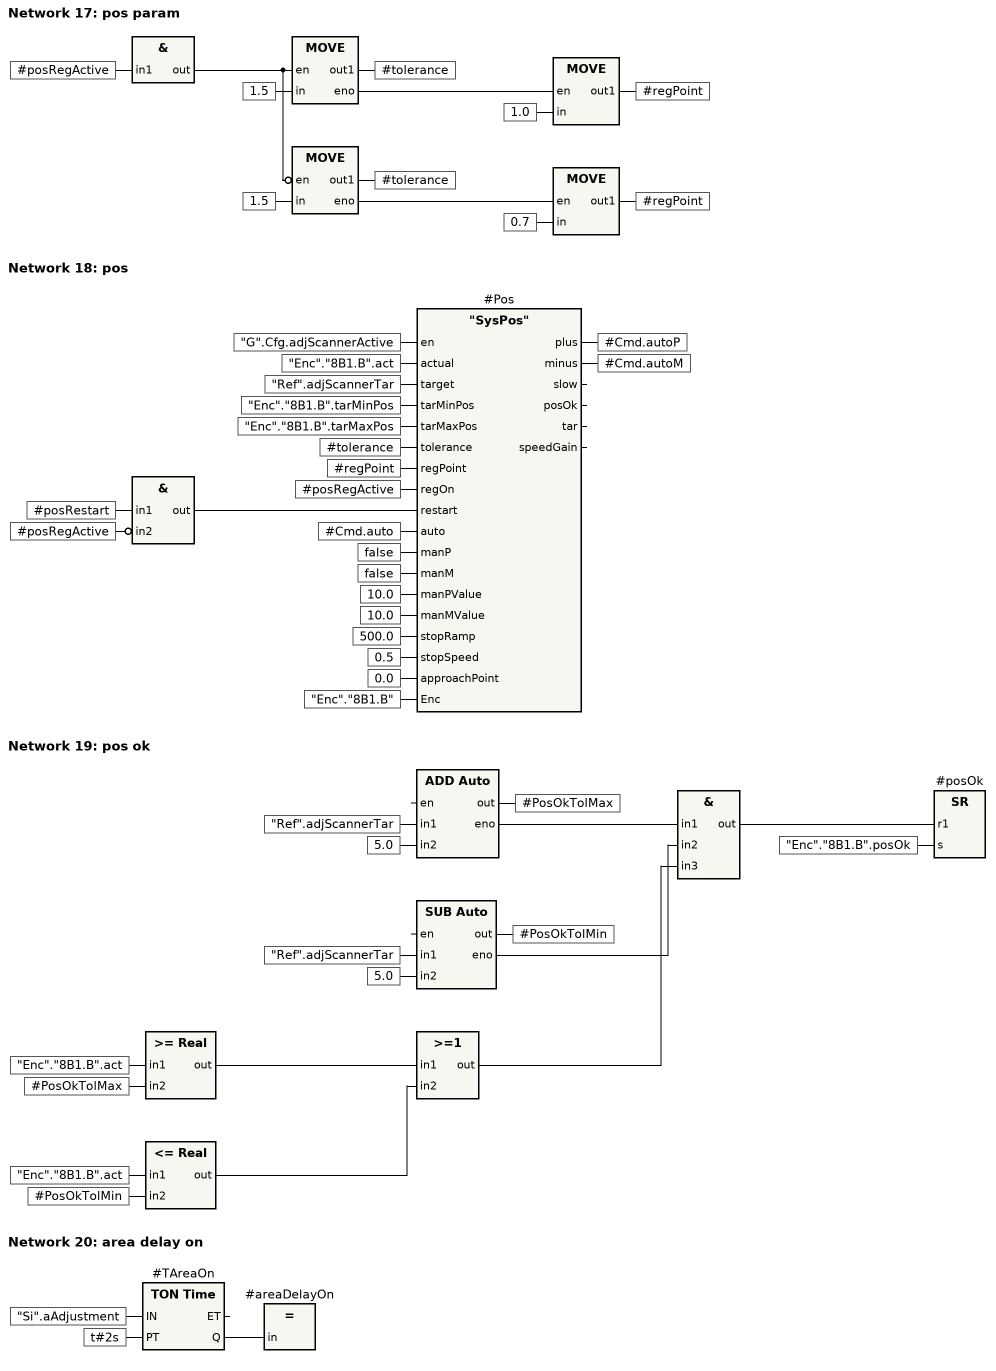
   IF #posRegActive THEN
       #tolerance := 1.5;
       #regPoint := 1.0;
   END_IF;
   IF NOT #posRegActive THEN
       #tolerance := 1.5;
       #regPoint := 0.7;
   END_IF;
END_REGION

REGION Network 18: pos
   IF "G".Cfg.adjScannerActive THEN
       #Pos(actual := "Enc"."8B1.B".act,   // "SysPos"
            target := "Ref".adjScannerTar,
            tarMinPos := "Enc"."8B1.B".tarMinPos,
            tarMaxPos := "Enc"."8B1.B".tarMaxPos,
            tolerance := #tolerance,
            regPoint := #regPoint,
            regOn := #posRegActive,
            restart := #posRestart AND NOT #posRegActive,
            auto := #Cmd.auto,
            manP := false,
            manM := false,
            manPValue := 10.0,
            manMValue := 10.0,
            stopRamp := 500.0,
            stopSpeed := 0.5,
            approachPoint := 0.0,
            Enc := "Enc"."8B1.B",
            plus => #Cmd.autoP,
            minus => #Cmd.autoM);
   END_IF;
END_REGION

REGION Network 19: pos ok
   #PosOkTolMax := "Ref".adjScannerTar + 5.0;
   #PosOkTolMin := "Ref".adjScannerTar - 5.0;
   IF "Enc"."8B1.B".posOk THEN
       #posOk := TRUE;   // SR flip-flop
   END_IF;
   IF ("Enc"."8B1.B".act >= #PosOkTolMax) OR ("Enc"."8B1.B".act <= #PosOkTolMin) THEN
       #posOk := FALSE;
   END_IF;
END_REGION

REGION Network 20: area delay on
   #TAreaOn(IN := "Si".aAdjustment, PT := t#2s);   // TON
   #areaDelayOn := #TAreaOn.Q;
END_REGION

REGION Network 21: motor
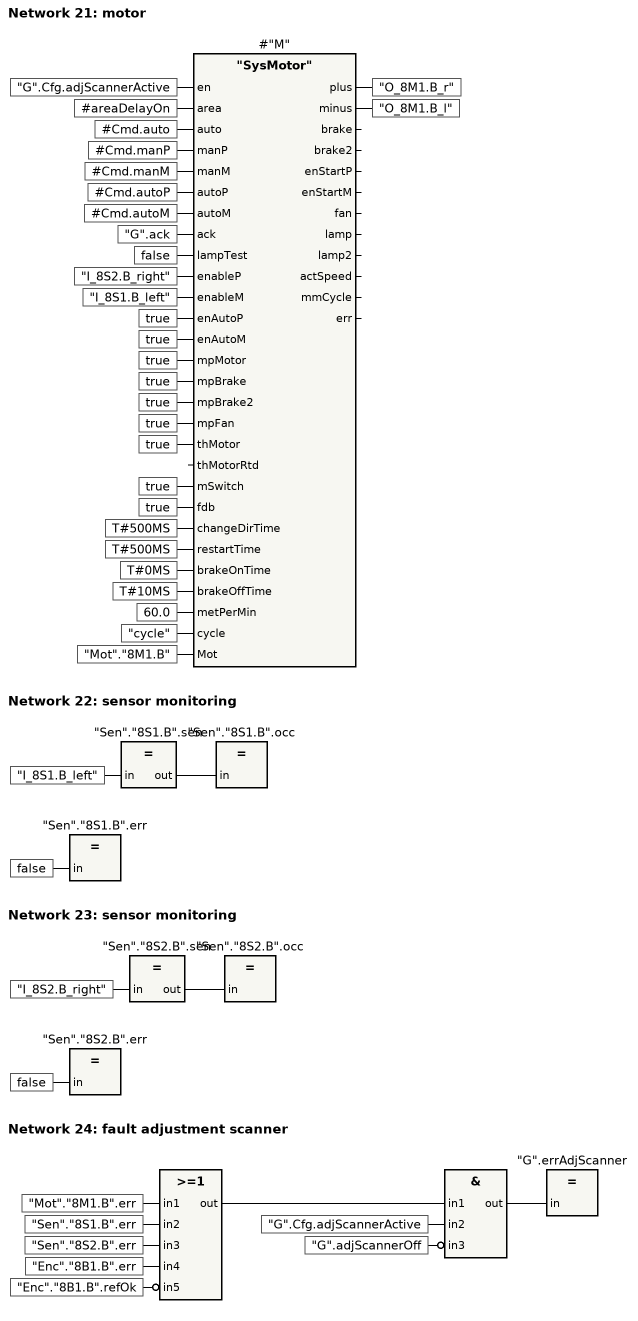
   IF "G".Cfg.adjScannerActive THEN
       #"M"(area := #areaDelayOn,   // "SysMotor"
            auto := #Cmd.auto,
            manP := #Cmd.manP,
            manM := #Cmd.manM,
            autoP := #Cmd.autoP,
            autoM := #Cmd.autoM,
            ack := "G".ack,
            lampTest := false,
            enableP := "I_8S2.B_right",
            enableM := "I_8S1.B_left",
            enAutoP := true,
            enAutoM := true,
            mpMotor := true,
            mpBrake := true,
            mpBrake2 := true,
            mpFan := true,
            thMotor := true,
            mSwitch := true,
            fdb := true,
            changeDirTime := T#500MS,
            restartTime := T#500MS,
            brakeOnTime := T#0MS,
            brakeOffTime := T#10MS,
            metPerMin := 60.0,
            cycle := "cycle",
            Mot := "Mot"."8M1.B",
            plus => "O_8M1.B_r",
            minus => "O_8M1.B_l");
   END_IF;
END_REGION

REGION Network 22: sensor monitoring
   "Sen"."8S1.B".sen := "I_8S1.B_left";
   "Sen"."8S1.B".occ := "I_8S1.B_left";
   "Sen"."8S1.B".err := false;
END_REGION

REGION Network 23: sensor monitoring
   "Sen"."8S2.B".sen := "I_8S2.B_right";
   "Sen"."8S2.B".occ := "I_8S2.B_right";
   "Sen"."8S2.B".err := false;
END_REGION

REGION Network 24: fault adjustment scanner
   "G".errAdjScanner := ("Mot"."8M1.B".err OR "Sen"."8S1.B".err OR "Sen"."8S2.B".err OR "Enc"."8B1.B".err OR NOT "Enc"."8B1.B".refOk) AND "G".Cfg.adjScannerActive AND NOT "G".adjScannerOff;
END_REGION

REGION Network 25 (SCL): data to pc
   IF "G".Cfg.adjScannerActive THEN
       "Ref".adjScannerAct := REAL_TO_DINT("Enc"."8B1.B".act * 10.0);
       "ComSd".Data.Scanner.ActualEncPos := "Enc"."8B1.B".encAct;
       IF "G".Cfg.modeBoardPassing = 2 THEN
           "ComSd".Data.Scanner.ActualPos := "Ref".adjScannerAct * -1;
           "ComSd".Data.Scanner.Plus := "Mot"."8M1.B".minus;
           "ComSd".Data.Scanner.Minus := "Mot"."8M1.B".plus;
       ELSE
           "ComSd".Data.Scanner.ActualPos := "Ref".adjScannerAct;
           "ComSd".Data.Scanner.Plus := "Mot"."8M1.B".plus;
           "ComSd".Data.Scanner.Minus := "Mot"."8M1.B".minus;
       END_IF;
       "ComSd".Data.Scanner.LimitSwitchMin := "Sen"."8S1.B".sen;
       "ComSd".Data.Scanner.LimitSwitchMax := "Sen"."8S2.B".sen;
       "ComSd".Data.Scanner.Err := "Mot"."8M1.B".err;
       "ComSd".Data.Scanner.ErrEnc := "Enc"."8B1.B".err;
       "ComSd".Data.Scanner.PosOk := ("Enc"."8B1.B".posOk AND #posRegActive) OR (#posOk AND NOT #posRegActive);
       "ComSd".Data.Scanner.refRun := "Enc"."8B1.B".refRun;
       "ComSd".Data.Scanner.refOk := "Enc"."8B1.B".refOk;
   ELSE
       "ComSd".Data.Scanner.ActualEncPos := 0;
       "ComSd".Data.Scanner.ActualPos := 0;
       "ComSd".Data.Scanner.LimitSwitchMin := FALSE;
       "ComSd".Data.Scanner.LimitSwitchMax := FALSE;
       "ComSd".Data.Scanner.Err := FALSE;
       "ComSd".Data.Scanner.ErrEnc := FALSE;
       "ComSd".Data.Scanner.PosOk := TRUE;
       "ComSd".Data.Scanner.Plus := FALSE;
       "ComSd".Data.Scanner.Minus := FALSE;
       "ComSd".Data.Scanner.refRun := FALSE;
       "ComSd".Data.Scanner.refOk := TRUE;
   END_IF;
END_REGION
END_FUNCTION_BLOCK

FUNCTION_BLOCK "SysBaluffBUS007F"   // FB4010, FBD
{ S7_Optimized_Access := 'TRUE' }
// stored: AutoNumber false, MemoryReserve 100, SetENOAutomatically false
   VAR_INPUT
      adrHW { ExternalAccessible := 'False'; ExternalVisible := 'False'; ExternalWritable := 'False'} : HW_IO;   // I/O adress HW / I/O adress
      adr { ExternalAccessible := 'False'; ExternalVisible := 'False'; ExternalWritable := 'False'} : Int;   // I/O adress
      slot { ExternalAccessible := 'False'; ExternalVisible := 'False'; ExternalWritable := 'False'} : Int;   // slot of io link module 1..4
      ack { ExternalAccessible := 'False'; ExternalVisible := 'False'; ExternalWritable := 'False'} : Bool;   // acknowledge
      startConfig { ExternalAccessible := 'False'; ExternalVisible := 'False'; ExternalWritable := 'False'} : Bool;
   END_VAR
   VAR_OUTPUT
      Measure { ExternalAccessible := 'False'; ExternalVisible := 'False'; ExternalWritable := 'False'} : Real;   // Actual measured value [mm] (-1= Read error)
      Scale { ExternalAccessible := 'False'; ExternalVisible := 'False'; ExternalWritable := 'False'} : Real;   // Scale -1 = 1/10mm
      ComOk { ExternalAccessible := 'False'; ExternalVisible := 'False'; ExternalWritable := 'False'} : Bool;   // communication ok
      ConfigOk { ExternalAccessible := 'False'; ExternalVisible := 'False'; ExternalWritable := 'False'} : Bool;   // configuration ok
      MeasureOk { ExternalAccessible := 'False'; ExternalVisible := 'False'; ExternalWritable := 'False'} : Bool;   // measuring ok
      Err { ExternalAccessible := 'False'; ExternalVisible := 'False'; ExternalWritable := 'False'} : Bool;   // Signal sensor error (1= Error)
      Warn { ExternalAccessible := 'False'; ExternalVisible := 'False'; ExternalWritable := 'False'} : Bool;   // Signal sensorwarning (1= Dirty)
      A1 { ExternalAccessible := 'False'; ExternalVisible := 'False'; ExternalWritable := 'False'} : Bool;   // Signal output 1 (1= Occ)
   END_VAR
   VAR_IN_OUT
      param : "TypeIOLinkParamArray";
   END_VAR
   VAR
      var { ExternalAccessible := 'False'; ExternalVisible := 'False'; ExternalWritable := 'False'} : Struct
         "bool" : Bool;
         "byte" : Byte;
         "word" : Word;
         "dword" : DWord;
         "int" : Int;
         "dint" : DInt;
         "real" : Real;
         s5time : S5Time;
         "time" : Time;
         hm : Array[1..50] of Bool;
         fm : Array[1..50] of Bool;
      END_STRUCT;
      Rd { ExternalAccessible := 'False'; ExternalVisible := 'False'; ExternalWritable := 'False'} : "TypeBaluffBUS007xRd";
      Data { ExternalAccessible := 'False'; ExternalVisible := 'False'; ExternalWritable := 'False'} : Struct
         Measure : Real;
         Scale : Real;
         ComOk : Bool;
         ConfigOk : Bool;
         MeasureOk : Bool;
         A1 : Bool;
         A2 : Bool;
         Warn : Bool;
         Err : Bool;
         ErrCom : Bool;
         ErrSensor : Bool;
         ErrConfig : Bool;
         WarnSensor : Bool;
      END_STRUCT;
      device { ExternalAccessible := 'False'; ExternalVisible := 'False'; ExternalWritable := 'False'} : "LIOLink_Device";
      statRecord { ExternalAccessible := 'False'; ExternalVisible := 'False'; ExternalWritable := 'False'} : Array[0..231] of Byte;
      cfgData { ExternalAccessible := 'False'; ExternalVisible := 'False'; ExternalWritable := 'False'} : Struct
         Index : Int;
         Subindex : Int;
         Len : Int;
         Value : "TypeIOLinkParamData";
      END_STRUCT;
      cfg { ExternalAccessible := 'False'; ExternalVisible := 'False'; ExternalWritable := 'False'} : Struct
         "Step" : Int;
         Done : Bool;
         Active : Bool;
         Err : Bool;
         Restart : Bool;
      END_STRUCT;
      T1 { ExternalAccessible := 'False'; ExternalVisible := 'False'; ExternalWritable := 'False'} : TON_TIME;
      cnt_i { ExternalAccessible := 'False'; ExternalVisible := 'False'; ExternalWritable := 'False'} : Int;
      cnt_y { ExternalAccessible := 'False'; ExternalVisible := 'False'; ExternalWritable := 'False'} : Int;
      cnt_x { ExternalAccessible := 'False'; ExternalVisible := 'False'; ExternalWritable := 'False'} : Int;
   END_VAR
   VAR_TEMP
      t_Data1 : Word;
      t_Data2 : Byte;
      t_Data3 : Byte;
      t_ENO : Bool;
   END_VAR
BEGIN

REGION Network 1 (SCL): info
   (*            
       Serie:          Baluff BUS007F  
       Type:           Baluff BUS M18M1-GPXI-03/025-S92G-511
       Range:          30..350mm
       Vendor ID:      888
       Device ID:      264209
       Input:          4 Byte
       Output:         0 Byte   

       Autor:          Alexander Kiebacher
       Datum:          05/2024
       Änderung:       05/2024
       Version:        1.0
       Lizenz:         Microtec

       Revisionen:     V1.0
   *)
END_REGION

REGION Network 2 (SCL): read data

   #t_Data1 := PEEK_WORD(area := 16#1, dbNumber := 0, byteOffset := #adr, ENO => #t_ENO);
   #t_Data2 := PEEK_BYTE(area := 16#1, dbNumber := 0, byteOffset := #adr + 2, ENO => #t_ENO);
   #t_Data3 := PEEK_BYTE(area := 16#1, dbNumber := 0, byteOffset := #adr + 3, ENO => #t_ENO);
   ENO := #t_ENO;
END_REGION

REGION Network 3 (SCL): read data - copy data
   // #Data.Scale := WORD_TO_SINT(SHR(IN := #t_Data2 AND 16#FF00, N := 8));
   // 
   // 0x80000008 –2147483640 Objekt zu nah
   // 0x7FFFFFF8 2147483640 Objekt zu weit
   // 0x7FFFFFFC 2147483644 Kein Signal

   IF ENO THEN

       #Rd.Measure := WORD_TO_INT(#t_Data1);
       #Rd.Scale := BYTE_TO_SINT(#t_Data2);

       #Rd.SCC1 := #t_Data3.%X0;

       // check communication
       #Data.MeasureOk := false;
       IF #Rd.Measure <> 0 THEN
           #Data.ComOk := true;
       ELSE
           #Data.ComOk := false;
       END_IF;

       IF #Rd.Measure = 32764 THEN             // no measurement data
           #Data.Measure := -1.0;
       ELSIF #Rd.Measure <= -32760 THEN        // out of measuring range (-)
           #Data.Measure := -1.0;
       ELSIF #Rd.Measure >= 32760 THEN         // out of measuring range (+)
           #Data.Measure := -1.0;
       ELSIF #Data.ComOk THEN
           #Data.Measure := INT_TO_REAL(#Rd.Measure) / 10.0;
           #Data.MeasureOk := true;
       END_IF;


       #Data.Scale := SINT_TO_REAL(#Rd.Scale);
       #Data.A1 := #Rd.SCC1;
       #Data.A2 := false;

   ELSE
       #Data.Measure := -1.0;
       #Data.Scale := 0.0;
       #Data.A1 := false;
       #Data.A2 := false;
       #Data.ComOk := false;

   END_IF;
END_REGION

REGION Network 5: reset fault / warning / reset faults
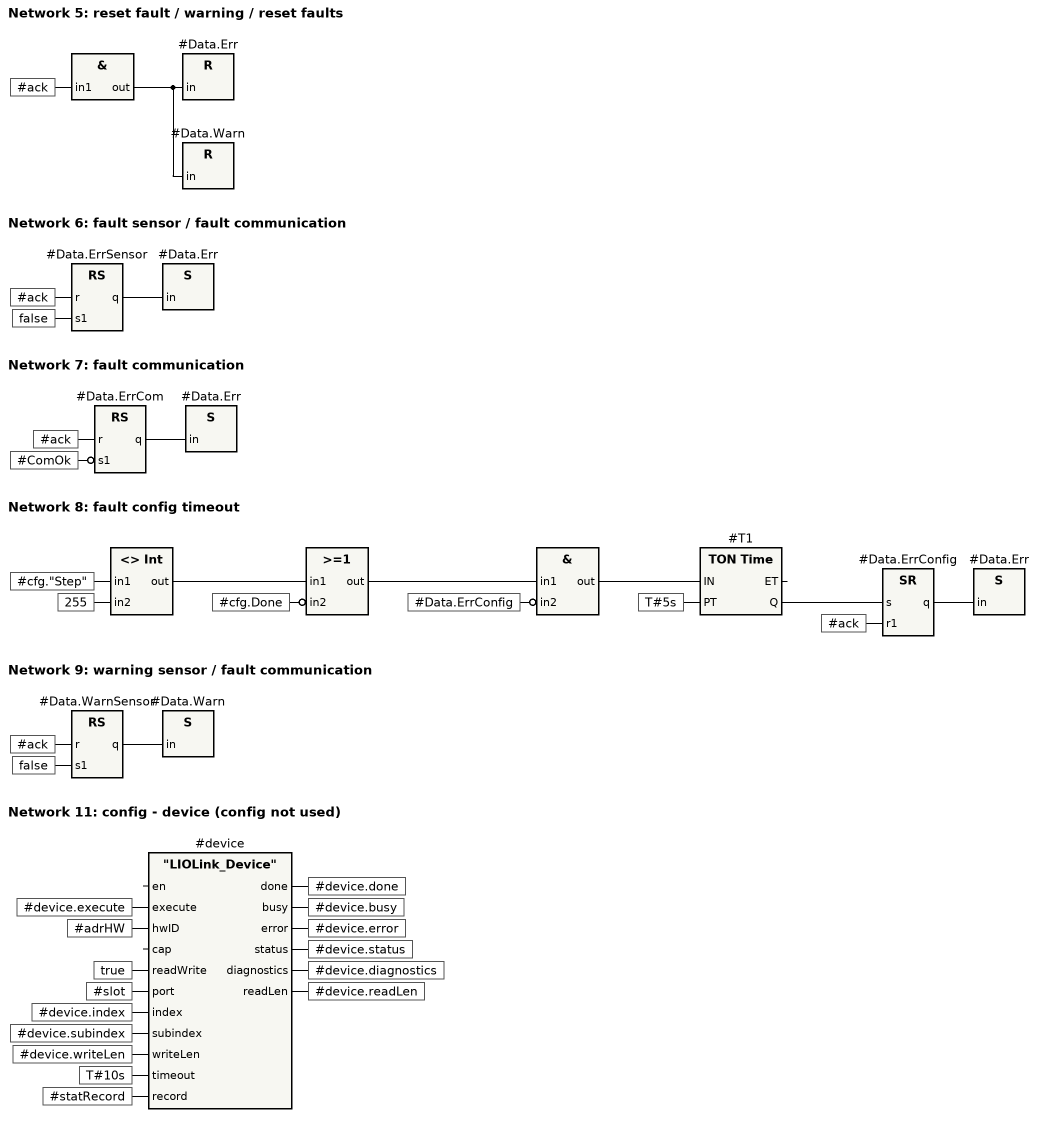
   IF #ack THEN
       #Data.Err := FALSE;
       #Data.Warn := FALSE;
   END_IF;
END_REGION

REGION Network 6: fault sensor / fault communication
   IF #ack THEN
       #Data.ErrSensor := FALSE;   // RS flip-flop
   END_IF;
   IF false THEN #Data.ErrSensor := TRUE; END_IF;
   IF #Data.ErrSensor THEN #Data.Err := TRUE; END_IF;
END_REGION

REGION Network 7: fault communication
   IF #ack THEN
       #Data.ErrCom := FALSE;   // RS flip-flop
   END_IF;
   IF NOT #ComOk THEN #Data.ErrCom := TRUE; END_IF;
   IF #Data.ErrCom THEN #Data.Err := TRUE; END_IF;
END_REGION

REGION Network 8: fault config timeout
   #T1(IN := ((#cfg."Step" <> 255) OR NOT #cfg.Done) AND NOT #Data.ErrConfig, PT := T#5s);   // TON
   IF #T1.Q THEN
       #Data.ErrConfig := TRUE;   // SR flip-flop
   END_IF;
   IF #ack THEN #Data.ErrConfig := FALSE; END_IF;
   IF #Data.ErrConfig THEN #Data.Err := TRUE; END_IF;
END_REGION

REGION Network 9: warning sensor / fault communication
   IF #ack THEN
       #Data.WarnSensor := FALSE;   // RS flip-flop
   END_IF;
   IF false THEN #Data.WarnSensor := TRUE; END_IF;
   IF #Data.WarnSensor THEN #Data.Warn := TRUE; END_IF;
END_REGION

REGION Network 11: config - device (config not used)
   #device(execute := #device.execute,   // "LIOLink_Device"
           hwID := #adrHW,
           readWrite := true,
           port := #slot,
           index := #device.index,
           subindex := #device.subindex,
           writeLen := #device.writeLen,
           timeout := T#10s,
           record := #statRecord,
           done => #device.done,
           busy => #device.busy,
           error => #device.error,
           status => #device.status,
           diagnostics => #device.diagnostics,
           readLen => #device.readLen);
END_REGION

REGION Network 12 (SCL): config - device (config not used)
   (* Invalid *)

   IF (#cfg.Step <= 0 OR #cfg.Step > 255 OR #Data.ErrConfig) THEN
       #cfg.Done := false;
       #cfg.Err := true;
       #cfg.Step := 1;
       #device.execute := false;
   END_IF;

   CASE #cfg.Step OF
       1:  (* Not configured or config request *)
           IF (NOT #cfg.Done OR #cfg.Restart) AND NOT #Data.ErrConfig THEN
               #cfg.Done := false;
               #cfg.Restart := false;
               #cfg.Err := true;
               #cfg.Step := 20;
               #cnt_i := 0;
               #device.execute := false;
           END_IF;

   (* Setup correct operation mode *)        
       20: (* Start config  *)

           #cfgData.Index := #param.Param[#cnt_i].Index;
           #cfgData.Subindex := #param.Param[#cnt_i].Subindex;
           #cfgData.Len := #param.Param[#cnt_i].Len;

           FOR #cnt_y := 0 TO (#cfgData.Len - 1) BY 1 DO
               #cfgData.Value.data[#cnt_y] := #param.Param[#cnt_i].Value.data[#cnt_y];
           END_FOR;

           #device.index := #cfgData.Index ;
           #device.subindex := #cfgData.Subindex ;
           #device.writeLen := #cfgData.Len;
           FOR #cnt_x := 0 TO (#cfgData.Len - 1) BY 1 DO
               #statRecord[#cnt_x] := #cfgData.Value.data[#cnt_x];
           END_FOR;

           #device.execute := false;
           #cfg.Step := 21;

       21: (* Start request *)
           #device.execute := true;
           #cfg.Step := 22;

       22: (*Wait for execution *)
           IF #device.done THEN
               #device.execute := false;
               IF #param.Param[#cnt_i + 1].Len <> 0 THEN
                   #cnt_i := #cnt_i + 1;
                   #cfg.Step := 20;
               ELSE
                   #cfg.Step := 255;
               END_IF;

           END_IF;
           IF #device.error THEN
               #device.execute := false;
               #cfg.Step := 20;
           END_IF;

   (* Setup done *)
       255:
           #cfg.Done := true;
           #cfg.Err := false;

           IF #cfg.Done AND #startConfig THEN
               #cfg.Done := false;
               #cfg.Err := true;
               #cfg.Step := 1;
               #device.execute := false;
               #Data.ErrConfig := false;
           END_IF;

   END_CASE;

   #cfg.Active := #cfg.Step > 10 AND #cfg.Step <255;

   #Data.ConfigOk := #cfg.Done;

   IF TRUE THEN

       #Data.ConfigOk := TRUE;
       #cfg.Done := TRUE;
       #cfg.Step := 255;

   END_IF;
END_REGION

REGION Network 13 (SCL): write outputs

   #Measure := #Data.Measure;
   #Scale := #Data.Scale;
   #ComOk := #Data.ComOk;
   #ConfigOk := #Data.ConfigOk;
   #MeasureOk := #Data.MeasureOk;
   #Err := #Data.Err;
   #Warn := #Data.Warn;
   #A1 := #Data.A1;
END_REGION
END_FUNCTION_BLOCK

FUNCTION "SysCal1x" : Void   // FC2010, FBD
TITLE = one point callibration, work only with encoder data structure
{ S7_Optimized_Access := 'TRUE' }
AUTHOR : MiCROTEC
VERSION : 1.0
// -2017.03 : Martin
// stored: AutoNumber false, SetENOAutomatically false
   VAR_INPUT
      p1Set : Bool;   // set calibration point 1
      p1Inc : DInt;   // callibration point 1 in increment
      p1Mm : Real;   // callibration point 1 in millimeter
      encAct : DInt;   // actual position encoder
      gain : Real;   // callibration gain
      limMin : Real;   // limit position minimum
      limMax : Real;   // limit position maximum
      ack : Bool;   // fault acknowledge
   END_VAR
   VAR_OUTPUT
      calGain : Real;   // callibration gain
      calOffset : Real;   // callibration offset
      act : Real;   // actual position
      err : Bool;   // fault
   END_VAR
   VAR_IN_OUT
      Enc : "TypeEncoder";
   END_VAR
   VAR_TEMP
      tempAct : Real;   // actual position
   END_VAR
BEGIN

REGION Network 1: save callibration point 1
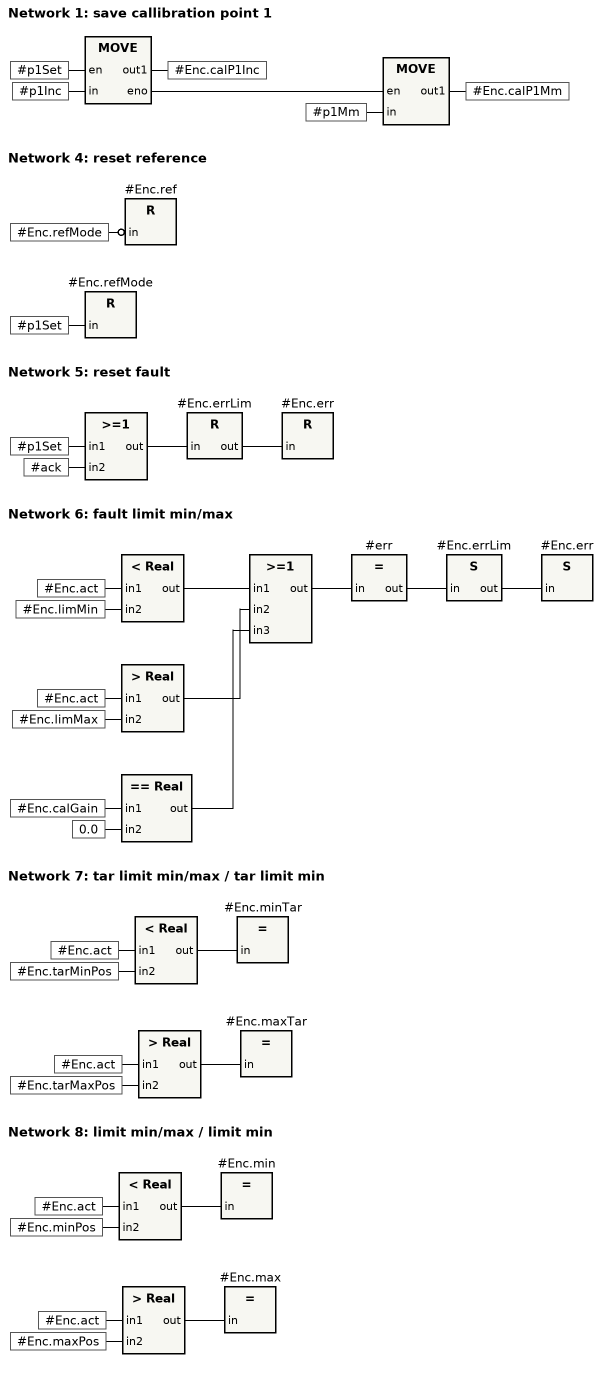
   // ENO of a box is taken as its EN; it also drops when the box reports an error
   IF #p1Set THEN
       #Enc.calP1Inc := #p1Inc;
       #Enc.calP1Mm := #p1Mm;
   END_IF;
END_REGION

REGION Network 2 (SCL): calculations
   #Enc.calGain := #gain;
   #Enc.calOffset := #Enc.calP1Mm - (DINT_TO_REAL(#Enc.calP1Inc) * #Enc.calGain);

   #Enc.act := (DINT_TO_REAL(#encAct - #Enc.calP1Inc) * #Enc.calGain) + #Enc.calP1Mm;
   #Enc.delta := DINT_TO_REAL(#Enc.deltaInc) * #Enc.calGain;
   #Enc.speed := #Enc.delta * 60.0 / "cycle";
END_REGION

REGION Network 3 (SCL): read/write values
   #Enc.limMin := #limMin;
   #Enc.limMax := #limMax;

   #calOffset := #Enc.calOffset;
   #calGain := #Enc.calGain;
   #act := #Enc.act;
END_REGION

REGION Network 4: reset reference
   IF NOT #Enc.refMode THEN #Enc.ref := FALSE; END_IF;
   IF #p1Set THEN #Enc.refMode := FALSE; END_IF;
END_REGION

REGION Network 5: reset fault
   IF #p1Set OR #ack THEN
       #Enc.errLim := FALSE;
       #Enc.err := FALSE;
   END_IF;
END_REGION

REGION Network 6: fault limit min/max
   #err := (#Enc.act < #Enc.limMin) OR (#Enc.act > #Enc.limMax) OR (#Enc.calGain = 0.0);
   IF #err THEN
       #Enc.errLim := TRUE;
       #Enc.err := TRUE;
   END_IF;
END_REGION

REGION Network 7: tar limit min/max / tar limit min
   #Enc.minTar := #Enc.act < #Enc.tarMinPos;
   #Enc.maxTar := #Enc.act > #Enc.tarMaxPos;
END_REGION

REGION Network 8: limit min/max / limit min
   #Enc.min := #Enc.act < #Enc.minPos;
   #Enc.max := #Enc.act > #Enc.maxPos;
END_REGION
END_FUNCTION

